IF ConveyorHasFault OR NOT SystemSafety.Safety_SystemEstopsOK THEN
	// Red light SOLID ON
	GVL_IO.LT_7221_Red := TRUE;
ELSE
	IF ConveyorHasWarn THEN
		// Orange Light SOLID ON
		GVL_IO.LT_7241_Yellow := TRUE;
	ELSE
		IF ConveyorInAuto THEN
			// Green Light SOLID ON
			GVL_IO.LT_7271_Green := TRUE;
		ELSE
			GVL_IO.LT_7271_Green := SysShrtPulseTmr.Output;
		END_IF
	END_IF
	IF GVL_IO.HornMainPanel THEN
		// Orange Light FLASHING ON
		GVL_IO.LT_7241_Yellow := SysShrtPulseTmr.Output;
	END_IF;
END_IF

// Initialise the Stack Light, only changing values as required
GVL_IO.LT_12161_Green := FALSE;
GVL_IO.LT_12131_Yellow := FALSE;
GVL_IO.LT_12121_Red := FALSE;
	
IF ConveyorHasFault OR NOT SystemSafety.Safety_SystemEstopsOK THEN
	// Red light SOLID ON
	GVL_IO.LT_12121_Red := TRUE;
ELSE
	IF ConveyorHasWarn THEN
		// Orange Light SOLID ON
		GVL_IO.LT_12131_Yellow := TRUE;
	ELSE
		IF ConveyorInAuto THEN
			// Green Light SOLID ON
			GVL_IO.LT_12161_Green := TRUE;
		ELSE
			GVL_IO.LT_12161_Green := SysShrtPulseTmr.Output;
		END_IF
	END_IF
	IF GVL_IO.HornMainPanel THEN
		// Orange Light FLASHING ON
		GVL_IO.LT_12131_Yellow := SysShrtPulseTmr.Output;
	END_IF;
END_IF

END_PROGRAM

// ---- POUs/FunctionBlocks/Utils/FB_SystemCntrl.TcPOU
FUNCTION_BLOCK FB_SystemCntrl

(* System Interlock and Event Set up,
	Uses Interlocks.
	Doesn't use Start Conditions or the horn delay  
	Uses Events
	
	This exists to allow the Interlock/Event descriptions and setup to be managed through the HMI
	and be easily setup as system faults.
*)
VAR_IN_OUT
	Sts_EquipState				: ST_EquipmentStatus;		// State Status
END_VAR
VAR_INPUT
	{attribute 'OPC.UA.DA' := '1'}
	In_o_EquipStatePB			: ST_StateCntrlPB;		// Hmi push buttons to change states
	In_p_EquipStatePB			: ST_StateCntrlPB;		// Other push buttons to change states
	{attribute 'OPC.UA.DA' := '1'}
	Cfg_EquipLabel				: STRING(20);		// Label of the equipment
	// Events
	In_SystemEvents				: UINT;		// Event that is specific to the instance of the solenoid/actuator
	Cfg_EquipEvntsArry			: ARRAY [0..15] OF ST_CfgEvents;
	
	// Interlocks that can be Instance Specific
	In_SystemIntlks				: UINT;		// Interlock that is specific to the instance of the solenoid/actuator
	Cfg_EquipIntlksArry		: ARRAY [0..15] OF ST_CfgEvents;		// Descriptions of the Interlock 
	
END_VAR
VAR_OUTPUT
	{attribute 'OPC.UA.DA' := '1'}
	Out_Auto					:	BOOL;	// Combine HMI and Other Start/Auto signals to issue a single START/AUTO command
	{attribute 'OPC.UA.DA' := '1'}
	Out_Stop					:	BOOL;	// Combine HMI and Other Stop signals to issue a single STOP command
	{attribute 'OPC.UA.DA' := '1'}
	Out_Reset					:	BOOL;	// Combine HMI and Other Reset signals to issue a single RESET command
	{attribute 'OPC.UA.DA' := '1'}
	Sts_All_Intlks_OK			: BOOL;		// Status bit to show that all interloks are good to Run 
	{attribute 'OPC.UA.DA' := '1'}
	Sts_FaultActive				: BOOL;	// Status Bit Showing that a fault is present (0= No Active Faults, 1= Fault Active)
	{attribute 'OPC.UA.DA' := '1'}
	Sts_WarnActive				: BOOL;	// Status Bit Showing that a warning is present (0= No Active Warnings, 1= Warning Active)
	{attribute 'OPC.UA.DA' := '1'}
	Sts_All_Evnts_OK			: BOOL;		// Status Bit Showing that ALL Events are OK to RUN (0= Event Present, 1= OK to Run)
	{attribute 'OPC.UA.DA' := '1'}
	Sts_IntlksArry				: ARRAY[0..15] OF ST_EventSts;		// Interlock status 0 to 15 Input
	{attribute 'OPC.UA.DA' := '1'}
	Sts_FaultsArry				: ARRAY[0..15] OF ST_EventSts;	// Status of each Fault Event State (0= OFF, 1=ON)
	{attribute 'OPC.UA.DA' := '1'}
	Sts_WarnsArry				: ARRAY[0..15] OF ST_EventSts;		// Status of each Warning Event State (0= OFF, 1=ON)
	{attribute 'OPC.UA.DA' := '1'}
	Sts_EvntsArry				: ARRAY[0..15] OF ST_EventSts; 	// Status of each Event State (0= OFF, 1=ON)
END_VAR
VAR
	System_fbIntrlks				: FB_Intlks_Latch;
	System_IntlksArry				: ARRAY[0..15] OF BOOL;
	System_EventManager				: FB_EventMngr;
	System_EventArry				: ARRAY[0..15] OF BOOL;
	System_LatchIgnore				: BOOL := FALSE;		// Put as a place holder for ease of future use
	System_LatchReset				: BOOL := FALSE;		//Put as a place holder for ease of future use
	System_IntlkBypassed			: ARRAY [0..15] OF BOOL;		//Put as a place holder for ease of future use
END_VAR

// Set Up inputs for interlocks that are specific for the configuration instance
System_IntlksArry[0] := In_SystemIntlks.0;
System_IntlksArry[1] := In_SystemIntlks.1; 
System_IntlksArry[2] := In_SystemIntlks.2;
System_IntlksArry[3] := In_SystemIntlks.3;
System_IntlksArry[4] := In_SystemIntlks.4;
System_IntlksArry[5] := In_SystemIntlks.5;
System_IntlksArry[6] := In_SystemIntlks.6;
System_IntlksArry[7] := In_SystemIntlks.7;
System_IntlksArry[8] := In_SystemIntlks.8;
System_IntlksArry[9] := In_SystemIntlks.9; 
System_IntlksArry[10] := In_SystemIntlks.10;
System_IntlksArry[11] := In_SystemIntlks.11;
System_IntlksArry[12] := In_SystemIntlks.12;
System_IntlksArry[13] := In_SystemIntlks.13;
System_IntlksArry[14] := In_SystemIntlks.14;
System_IntlksArry[15] := In_SystemIntlks.15;
	
// Call Interlock block
System_fbIntrlks(
	In_Intlks:= System_IntlksArry,
	CFG_IntlksArry:= Cfg_EquipIntlksArry, 
	HMI_LatchIgnore:= System_LatchIgnore, 
	HMI_LatchReset:= System_LatchReset, 
	All_Intlk_OK=> Sts_All_Intlks_OK, 
	STS_Intlks=> Sts_IntlksArry);
	
System_EventArry[0]:= In_SystemEvents.0;
System_EventArry[1]:= In_SystemEvents.1;
System_EventArry[2]:= In_SystemEvents.2;
System_EventArry[3]:= In_SystemEvents.3;
System_EventArry[4]:= In_SystemEvents.4;
System_EventArry[5]:= In_SystemEvents.5;
System_EventArry[6]:= In_SystemEvents.6;
System_EventArry[7]:= In_SystemEvents.7;
System_EventArry[8]:= In_SystemEvents.8;
System_EventArry[9]:= In_SystemEvents.9;
System_EventArry[10]:= In_SystemEvents.10;
System_EventArry[11]:= In_SystemEvents.11;
System_EventArry[12]:= In_SystemEvents.12;
System_EventArry[13]:= In_SystemEvents.13;
System_EventArry[14]:= In_SystemEvents.14;
System_EventArry[15]:= In_SystemEvents.15;

// Event Manager
System_EventManager(
	sEquipStateCntrlSts := Sts_EquipState.Sts_EquipmentState,
	In_EventsArry := System_EventArry ,  
	CFG_EvntsArry:= Cfg_EquipEvntsArry, 
	HMI_LatchReset:= In_o_EquipStatePB.ResetPB OR In_p_EquipStatePB.ResetPB,
	Out_FaultActive=> Sts_FaultActive, 
	Out_WarnActive=> Sts_WarnActive, 
	Sts_All_Evnts_OK=> Sts_All_Evnts_OK, 
	Sts_FaultsArry=> Sts_FaultsArry, 
	Sts_WarnsArry=> Sts_WarnsArry, 
	Sts_EvntsArry=> Sts_EvntsArry);

// Activate the Out_ variables
Out_Auto := In_o_EquipStatePB.AutoPB OR In_p_EquipStatePB.AutoPB;
Out_Stop := In_o_EquipStatePB.StopPB OR In_p_EquipStatePB.StopPB;
Out_Reset := In_o_EquipStatePB.ResetPB OR In_p_EquipStatePB.ResetPB;

// Populate the Sts Output Variables
Sts_EquipState.Sts_EquipmentState.CrntState := 1;
Sts_EquipState.Sts_All_Intlks_OK  := Sts_All_Intlks_OK;
Sts_EquipState.Sts_All_Evnts_OK  := Sts_All_Evnts_OK;
Sts_EquipState.Sts_FaultActive := Sts_FaultActive;
Sts_EquipState.Sts_WarnActive := Sts_WarnActive;

END_FUNCTION_BLOCK

// ---- POUs/SystemSafety.TcPOU
PROGRAM SystemSafety
VAR
	{attribute 'OPC.UA.DA' := '1'}
	System_SafetyState : ST_SafetyState;
	{attribute 'OPC.UA.DA' := '1'}

	{attribute 'OPC.UA.DA' := '1'}
	Safety_SystemEstopsOK AT %I* : BOOL;
	{attribute 'OPC.UA.DA' := '1'}
	Safety_PanelEstop AT %I* : BOOL;
	{attribute 'OPC.UA.DA' := '1'}
	ZoneSafe_EDM AT %I*: BOOL; 
	{attribute 'OPC.UA.DA' := '1'}
	SecondFloorShaft_Estop_OK AT %I* : BOOL;
	{attribute 'OPC.UA.DA' := '1'}
	ThirdFloorShaft_Estop_OK AT %I* : BOOL;
END_VAR

// Set System Safety Variables 
System_SafetyState.ErrAck := System.Safety_Reset;
System_SafetyState.CommErrAck := System.Safety_Reset;
System_SafetyState.Reset := System.Safety_Reset;
System_SafetyState.Run := TRUE;

END_PROGRAM

// ---- POUs/FunctionBlocks/VFD/Functions/VFD.TcPOU
FUNCTION_BLOCK VFD
FUNCTION_BLOCK VFD
VAR_INPUT
	RunVelocity				: INT;
	RunRequest				: BOOL;
	PLCFault				: BOOL;
	Reset					: BOOL;
	VelocityThreshold		: INT;
END_VAR
VAR_OUTPUT
	ActualVelocity 	AT %I* 	: INT;
	StatusWord		AT %I* 	: UINT;
	Run_OK					: BOOL;
	STO_Active				: BOOL;
	IsRunning				: BOOL;
	IsFaulted 				: BOOL;
END_VAR
VAR
	VFD_State				: DriveState;
	ControlWord 	AT %Q* 	: UINT;
	TargetVelocity 	AT %Q*	: INT;
	StatusWordFiltered		: UINT;
END_VAR
VAR CONSTANT
	SAFETY_TORQUE_OFF_ACTIVE : INT := 15;
END_VAR

StatusWordFiltered := StatusWord AND 16#006F;

VFD_State(StatusWord := StatusWordFiltered, Run_Drive := RunRequest, ControlWord => ControlWord, PLCFault := PLCFault, ResetFault := Reset);

IF Reset THEN
	Reset := FALSE;
END_IF

Run_OK := (StatusWordFiltered = Drive_State.READY_TO_SWITCH_ON) OR (StatusWordFiltered = Drive_State.SWITCHED_ON) OR (StatusWordFiltered = Drive_State.OPERATION_ENABLED);

IF StatusWordFiltered = Drive_State.OPERATION_ENABLED THEN
	TargetVelocity := RunVelocity;
ELSE
	TargetVelocity := 0;	
END_IF

STO_Active := StatusWord.SAFETY_TORQUE_OFF_ACTIVE;
 
IsRunning := ActualVelocity >= VelocityThreshold;
IsFaulted := VFD_State.Fault;

END_FUNCTION_BLOCK

// ---- POUs/CommStatus.TcPOU
PROGRAM CommStatus
VAR
	In_Dummy		:	BOOL;	// Replace per function call with IO point

	DebounceOnTime:	TIME := T#500MS;     // Default Value	
	DebounceOffTime:	TIME := T#1S;     // Default Value
		
	RIO1181_CommFault: FB_DigDebnce;	// Remote IO Block 1181 Communication Fault
	RIO4172_CommFault: FB_DigDebnce;	// Remote IO Block 4172 Communication Fault
	RIO5151_CommFault: FB_DigDebnce;	// Remote IO Block 5151 Communication Fault
	RIO6171_CommFault: FB_DigDebnce;	// Remote IO Block 6171 Communication Fault
	RIO7161_CommFault: FB_DigDebnce;	// Remote IO Block 7161 Communication Fault
	RIO8181_CommFault: FB_DigDebnce;	// Remote IO Block 8181 Communication Fault
	RIO11141_CommFault: FB_DigDebnce;	// Remote IO Block 11141 Communication Fault	
	RIO12171_CommFault: FB_DigDebnce;	// Remote IO Block 12171 Communication Fault
	RIO15181_CommFault: FB_DigDebnce;	// Remote IO Block 15181 Communication Fault
	RIO16171_CommFault: FB_DigDebnce;	// Remote IO Block 16171 Communication Fault
	
	BCR_S6040_01_CommFault: FB_DigDebnce;;		// Bar Code Reader 6040_01 Communication Fault
	BCR_S7004_01_CommFault: FB_DigDebnce;;		// Bar Code Reader 7004_01 Communication Fault
	
	Ethernet_CommFault: FB_DigDebnce;;		// Ethernet Adapter Status Communication Fault
	
END_VAR

// Remote IO Blocks --------------------
RIO1181_CommFault(
	In:= GVL_IO.RIO1181_WcState, 
	CFG_OKState:= 0, 
	CFG_OnDlyTime:= DebounceOnTime, 
	CFG_OffDlyTime:= DebounceOffTime, 
	In_Sim:= , 
	);
	
RIO4172_CommFault(
	In:= GVL_IO.RIO4172_WcState, 
	CFG_OKState:= 0, 
	CFG_OnDlyTime:= DebounceOnTime, 
	CFG_OffDlyTime:= DebounceOffTime, 
	In_Sim:= , 
	);

RIO5151_CommFault(
	In:= GVL_IO.RIO5151_WcState, 
	CFG_OKState:= 0, 
	CFG_OnDlyTime:= DebounceOnTime, 
	CFG_OffDlyTime:= DebounceOffTime, 
	In_Sim:= , 
	);

RIO6171_CommFault(
	In:= GVL_IO.RIO6171_WcState, 
	CFG_OKState:= 0, 
	CFG_OnDlyTime:= DebounceOnTime, 
	CFG_OffDlyTime:= DebounceOffTime, 
	In_Sim:= , 
	);
	
RIO7161_CommFault(
	In:= GVL_IO.RIO7161_WcState, 
	CFG_OKState:= 0, 
	CFG_OnDlyTime:= DebounceOnTime, 
	CFG_OffDlyTime:= DebounceOffTime, 
	In_Sim:= , 
	);
	
RIO8181_CommFault(
	In:= GVL_IO.RIO8181_WcState, 
	CFG_OKState:= 0, 
	CFG_OnDlyTime:= DebounceOnTime, 
	CFG_OffDlyTime:= DebounceOffTime, 
	In_Sim:= , 
	);
	
RIO11141_CommFault(
	In:= GVL_IO.RIO11141_WcState, 
	CFG_OKState:= 0, 
	CFG_OnDlyTime:= DebounceOnTime, 
	CFG_OffDlyTime:= DebounceOffTime, 
	In_Sim:= , 
	);
	
RIO11141_CommFault(
	In:= GVL_IO.RIO11141_WcState, 
	CFG_OKState:= 0, 
	CFG_OnDlyTime:= DebounceOnTime, 
	CFG_OffDlyTime:= DebounceOffTime, 
	In_Sim:= , 
	);
	
RIO12171_CommFault(
	In:= GVL_IO.RIO12171_WcState, 
	CFG_OKState:= 0, 
	CFG_OnDlyTime:= DebounceOnTime, 
	CFG_OffDlyTime:= DebounceOffTime, 
	In_Sim:= , 
	);
	
RIO15181_CommFault(
	In:= GVL_IO.RIO15181_WcState, 
	CFG_OKState:= 0, 
	CFG_OnDlyTime:= DebounceOnTime, 
	CFG_OffDlyTime:= DebounceOffTime, 
	In_Sim:= , 
	);
	
RIO16171_CommFault(
	In:= GVL_IO.RIO16171_WcState, 
	CFG_OKState:= 0, 
	CFG_OnDlyTime:= DebounceOnTime, 
	CFG_OffDlyTime:= DebounceOffTime, 
	In_Sim:= , 
	);

// Bar Code Readers --------------------	
BCR_S6040_01_CommFault(
	In:= BarCodeReaders.BCR_S6040_01.Out_DeviceState = 0, 
	CFG_OKState:= 1, 
	CFG_OnDlyTime:= DebounceOnTime, 
	CFG_OffDlyTime:= DebounceOffTime, 
	In_Sim:= , 
	);
BCR_S7004_01_CommFault(
	In:= BarCodeReaders.BCR_S7004_01.Out_DeviceState = 0, 
	CFG_OKState:= 1, 
	CFG_OnDlyTime:= DebounceOnTime, 
	CFG_OffDlyTime:= DebounceOffTime, 
	In_Sim:= , 
	);
	
// Ethernet Controller	
Ethernet_CommFault(
	In:= GVL_IO.EthernetAdapter_State = 0, 
	CFG_OKState:= 1, 
	CFG_OnDlyTime:= DebounceOnTime, 
	CFG_OffDlyTime:= DebounceOffTime, 
	In_Sim:= , 
	);

END_PROGRAM

// ---- POUs/FunctionBlocks/Utils/Filters/FB_DigDebnce.TcPOU
(*
Function Block to filter the ON and OFF of a digital input In
The normal OK state can be configured with CFG_OKState
The Times for the On and Off delays are configured by CFG_OnDlyTime and CFG_OffDlyTime
and can be simulated using the In_Sim input
If the input In goes true the output OutOnFltrd is set to true after the on delay time has elapsed
If the input In goes false the output CFG_OffDlyTime will be held on until the off delay time has elapsed
The output OutOnOffFltrd is delayed for both on and off as described above
The status outputs Sts_OnDlyActive and Sts_OffDlyActive show that the delays are active
*)
FUNCTION_BLOCK FB_DigDebnce
VAR_INPUT
	In:	BOOL;	// Digital Input
	CFG_OKState:	BOOL;		// The OK or ON State of the Input (0 or 1)
	CFG_OnDlyTime:	TIME;		// Time to delay Output turning On after Input is On
	CFG_OffDlyTime:	TIME;		// Time to delay Output turning Off after Input is Off
	In_Sim:	BOOL;		// Simulation Input Bit acts just like the input but can be forced from the program for testing
END_VAR
VAR_OUTPUT
	{attribute 'OPC.UA.DA' := '1'}
	Out:	BOOL;		// Output Based on ON or OK state
	OutOnFltrd:	BOOL;		// ON filtered Only Output
	OutOffFltrd:	BOOL;		// Off filtered Only OutPut
	OutOnOffFltrd:	BOOL;		// Both On and Off Filtered Output 
	Sts_OnDlyActive: BOOL;
	Sts_OffDlyActive: BOOL;
	Sts_OnOffDlyActive: BOOL;
END_VAR
VAR
	OnDly_Ton: TON;
	OffDlyTof: TOF;
	OnOffDlyTof: TOF;
	OnOffDly_SR: SR;
	
END_VAR

// Compare to normal ON state
Out := (In OR In_Sim) XOR CFG_OKState;

// Setup On Delay
OnDly_Ton(IN:= Out, PT:= CFG_OnDlyTime , Q=> OutOnFltrd , ET=> );
Sts_OnDlyActive := Out <> OutOnFltrd;

//Setup Off Delay
OffDlyTof(IN:= Out , PT:= CFG_OffDlyTime , Q=> OutOffFltrd , ET=> );
Sts_OffDlyActive := Out <> OutOffFltrd;

//Setup Both On and Off Delayed
//OnOffDlyTof(IN:= OutOnFltrd , PT:= CFG_OffDlyTime , Q=> OutOnOffFltrd , ET=> );
OnOffDly_SR(SET1 := OutOnFltrd, RESET := (NOT OffDlyTof.Q), Q1 => OutOnOffFltrd);
Sts_OnOffDlyActive := Out <> OutOnOffFltrd;

END_FUNCTION_BLOCK

// ---- POUs/ProxSensors.TcPOU
PROGRAM ProxSensors
VAR
	DebounceOnTime:	TIME := T#5MS;     // Default Value
	DebounceOffTime:	TIME := T#500MS;     // Default Value
	JamDetectTime:	TIME := T#5S;     // Default Value

	
	In_PX_1281_Extended AT %I* : BOOL;      // Mapped IO input for PX
	PX_1281_Extended:  FB_DigDebnce;		// P6020 POWER TRANSFER EXTENDED PROX
//----------------------------------------GR6040_01--------------------------------------------------------------
	In_PX_6241_Retracted AT %I* : BOOL;      // Mapped IO input for PX
	PX_6241_Retracted:  FB_DigDebnce;		// GR6040-01 "D" GRIPPER RETRACTED PROX

	In_PX_6261_Extended AT %I* : BOOL;      // Mapped IO input for PX
	PX_6261_Extended:  FB_DigDebnce;		// GR6040-01 "D" GRIPPER EXTENDED PROX
//----------------------------------------GR6040_02--------------------------------------------------------------
	In_PX_6121_Retracted AT %I* : BOOL;      // Mapped IO input for PX
	PX_6121_Retracted:  FB_DigDebnce;		// GR6040-02 "D" GRIPPER RETRACTED PROX

	In_PX_6151_Extended AT %I* : BOOL;      // Mapped IO input for PX
	PX_6151_Extended:  FB_DigDebnce;		// GR6040-02 "D" GRIPPER EXTENDED PROX
//----------------------------------------PI6040_01--------------------------------------------------------------
	In_PX_6122_Retracted AT %I* : BOOL;      // Mapped IO input for PX
	PX_6122_Retracted:  FB_DigDebnce;		// PI6040-01 "D" GRIPPER RETRACTED PROX

	In_PX_6152_Extended AT %I* : BOOL;      // Mapped IO input for PX
	PX_6152_Extended:  FB_DigDebnce;		// PI6040-01 "D" GRIPPER EXTENDED PROX
//----------------------------------------PU6040_01--------------------------------------------------------------
	In_PX_7271_Retracted AT %I* : BOOL;      // Mapped IO input for PX
	PX_7271_Retracted:  FB_DigDebnce;		// PU6040-01 PUSH DIVERT RETRACTED PROX

	In_PX_7301_Extended AT %I* : BOOL;      // Mapped IO input for PX
	PX_7301_Extended:  FB_DigDebnce;		// PU6040-01 PUSH DIVERT EXTENDED PROX
//----------------------------------------PU6040_02--------------------------------------------------------------
	In_PX_7122_Retracted AT %I* : BOOL;      // Mapped IO input for PX
	PX_7122_Retracted:  FB_DigDebnce;		// PU6040-02 PUSH DIVERT RETRACTED PROX

	In_PX_7151_Extended AT %I* : BOOL;      // Mapped IO input for PX
	PX_7151_Extended:  FB_DigDebnce;		// PU6040-02 PUSH DIVERT EXTENDED PROX
//----------------------------------------PU6040_03--------------------------------------------------------------
	In_PX_8321_Retracted AT %I* : BOOL;      // Mapped IO input for PX
	PX_8321_Retracted:  FB_DigDebnce;		// PU6040-03 PUSH DIVERT RETRACTED PROX

	In_PX_8291_Extended AT %I* : BOOL;      // Mapped IO input for PX
	PX_8291_Extended:  FB_DigDebnce;		// PU6040-03 PUSH DIVERT EXTENDED PROX
//----------------------------------------PU6040_04--------------------------------------------------------------	
	In_PX_8091_Retracted AT %I* : BOOL;      // Mapped IO input for PX
	PX_8091_Retracted:  FB_DigDebnce;		// PU6040-04 PUSH DIVERT RETRACTED PROX

	In_PX_8121_Extended AT %I* : BOOL;      // Mapped IO input for PX
	PX_8121_Extended:  FB_DigDebnce;		// PU6040-04 PUSH DIVERT EXTENDED PROX

//------------------------------------------------------------------------------------------------------
	In_PX_16231_Extended AT %I* : BOOL;      // Mapped IO input for PX
	PX_16231_Extended:  FB_DigDebnce;		// P7035 POWER TRANSFER EXTENDED PROX

END_VAR

//----------------------------------------P6020--------------------------------------------------------------
// P6020 POWER TRANSFER Extended
PX_1281_Extended(
	In:= In_PX_1281_Extended,
	CFG_OKState:= 0,
	CFG_OnDlyTime:= DebounceOnTime,
	CFG_OnDlyTime:= DebounceOffTime,
	In_Sim:= 
	);
//----------------------------------------GR6040_01--------------------------------------------------------------
// GR6040-01 "D" GRIPPER Retracted
PX_6241_Retracted(
	In:= In_PX_6241_Retracted,
	CFG_OKState:= 0,
	CFG_OnDlyTime:= DebounceOnTime,
	CFG_OnDlyTime:= DebounceOffTime,
	In_Sim:= 
	);

// GR6040-01 "D" GRIPPER Extended
PX_6261_Extended(
	In:= In_PX_6261_Extended,
	CFG_OKState:= 0,
	CFG_OnDlyTime:= DebounceOnTime,
	CFG_OnDlyTime:= DebounceOffTime,
	In_Sim:= 
	);
//----------------------------------------GR6040_02--------------------------------------------------------------
// GR6040-02 "D" GRIPPER Retracted
PX_6121_Retracted(
	In:= In_PX_6121_Retracted,
	CFG_OKState:= 0,
	CFG_OnDlyTime:= DebounceOnTime,
	CFG_OnDlyTime:= DebounceOffTime,
	In_Sim:= 
	);

// GR6040-02 "D" GRIPPER Extended
PX_6151_Extended(
	In:= In_PX_6151_Extended,
	CFG_OKState:= 0,
	CFG_OnDlyTime:= DebounceOnTime,
	CFG_OnDlyTime:= DebounceOffTime,
	In_Sim:= 
	);
//----------------------------------------PI6040_01--------------------------------------------------------------
// PI6040-01 "D" GRIPPER Retracted
PX_6122_Retracted(
	In:= In_PX_6122_Retracted,
	CFG_OKState:= 0,
	CFG_OnDlyTime:= DebounceOnTime,
	CFG_OnDlyTime:= DebounceOffTime,
	In_Sim:= 
	);

// PI6040-01 "D" GRIPPER Extended
PX_6152_Extended(
	In:= In_PX_6152_Extended,
	CFG_OKState:= 0,
	CFG_OnDlyTime:= DebounceOnTime,
	CFG_OnDlyTime:= DebounceOffTime,
	In_Sim:= 
	);
//----------------------------------------PU6040_01--------------------------------------------------------------
// PU6040-01 PUSH DIVERT Retracted
PX_7271_Retracted(
	In:= In_PX_7271_Retracted,
	CFG_OKState:= 0,
	CFG_OnDlyTime:= DebounceOnTime,
	CFG_OnDlyTime:= DebounceOffTime,
	In_Sim:= 
	);

// PU6040-01 PUSH DIVERT Extended
PX_7301_Extended(
	In:= In_PX_7301_Extended,
	CFG_OKState:= 0,
	CFG_OnDlyTime:= DebounceOnTime,
	CFG_OnDlyTime:= DebounceOffTime,
	In_Sim:= 
	);
//----------------------------------------PU6040_02--------------------------------------------------------------
// PU6040-02 PUSH DIVERT Retracted
PX_7122_Retracted(
	In:= In_PX_7122_Retracted,
	CFG_OKState:= 0,
	CFG_OnDlyTime:= DebounceOnTime,
	CFG_OnDlyTime:= DebounceOffTime,
	In_Sim:= 
	);

// PU6040-02 PUSH DIVERT Extended
PX_7151_Extended(
	In:= In_PX_7151_Extended,
	CFG_OKState:= 0,
	CFG_OnDlyTime:= DebounceOnTime,
	CFG_OnDlyTime:= DebounceOffTime,
	In_Sim:= 
	);
//----------------------------------------PU6040_03--------------------------------------------------------------	
	// PU6040-03 PUSH DIVERT Retracted
PX_8321_Retracted(
	In:= In_PX_8321_Retracted,
	CFG_OKState:= 0,
	CFG_OnDlyTime:= DebounceOnTime,
	CFG_OnDlyTime:= DebounceOffTime,
	In_Sim:= 
	);

// PU6040-03 PUSH DIVERT Extended
PX_8291_Extended(
	In:= In_PX_8291_Extended,
	CFG_OKState:= 0,
	CFG_OnDlyTime:= DebounceOnTime,
	CFG_OnDlyTime:= DebounceOffTime,
	In_Sim:= 
	);
//----------------------------------------PU6040_04--------------------------------------------------------------
// PU6040-04 PUSH DIVERT Retracted
PX_8091_Retracted(
	In:= In_PX_8091_Retracted,
	CFG_OKState:= 0,
	CFG_OnDlyTime:= DebounceOnTime,
	CFG_OnDlyTime:= DebounceOffTime,
	In_Sim:= 
	);
	
// PU6040-04 PUSH DIVERT Extended
PX_8121_Extended(
	In:= In_PX_8121_Extended,
	CFG_OKState:= 0,
	CFG_OnDlyTime:= DebounceOnTime,
	CFG_OnDlyTime:= DebounceOffTime,
	In_Sim:= 
	);
//----------------------------------------P7035--------------------------------------------------------------
// P7035 POWER TRANSFER Extended
PX_16231_Extended(
	In:= In_PX_16231_Extended,
	CFG_OKState:= 0,
	CFG_OnDlyTime:= DebounceOnTime,
	CFG_OnDlyTime:= DebounceOffTime,
	In_Sim:= 
	);

END_PROGRAM

// ---- POUs/Solenoids.TcPOU
PROGRAM Solenoids

VAR
	 nEquipIndex:	DINT := 0;	// Dummy Equipment Index for Non reporting equipment
//----------------------------------------GR6040_02--------------------------------------------------------------
   cfgGR6040_02Label:	STRING(20) :=  'GR6040_02';
   cfgGR6040_02ExtendTODetectTime:	TIME := T#5S;
   cfgGR6040_02RetractTODetectTime:	TIME := T#5S;
   GR6040_02			: FB_Solenoid_SA;
   GR6040_02_StatePB	: ST_StateCntrlPB;
   GR6040_02_Status	: ST_EquipmentStatus;		// Gripper State 

//----------------------------------------GR6040_01--------------------------------------------------------------
   cfgGR6040_01Label:	STRING(20) :=  'GR6040_01';
   cfgGR6040_01ExtendTODetectTime:	TIME := T#5S;
   cfgGR6040_01RetractTODetectTime:	TIME := T#5S;
   GR6040_01			: FB_Solenoid_SA;
   GR6040_01_StatePB	: ST_StateCntrlPB;
   GR6040_01_Status	: ST_EquipmentStatus;		// Gripper State 

//----------------------------------------PI6040_01--------------------------------------------------------------
   cfgPI6040_01Label:	STRING(20) :=  'PI6040_01';
   cfgPI6040_01ExtendTODetectTime:	TIME := T#5S;
   cfgPI6040_01RetractTODetectTime:	TIME := T#5S;
   PI6040_01			: FB_Solenoid_DA;
   PI6040_01_StatePB	: ST_StateCntrlPB;
   PI6040_01_Status	: ST_EquipmentStatus;		// Gripper State 

//----------------------------------------PU6040_01--------------------------------------------------------------
   cfgPU6040_01Label:	STRING(20) :=  'PU6040_01';
   cfgPU6040_01ExtendTODetectTime:	TIME := T#5S;
   cfgPU6040_01RetractTODetectTime:	TIME := T#5S;
   PU6040_01			: FB_Solenoid_SA;
   PU6040_01_StatePB	: ST_StateCntrlPB;
   PU6040_01_Status	: ST_EquipmentStatus;		// Gripper State 

//----------------------------------------PU6040_02--------------------------------------------------------------
   cfgPU6040_02Label:	STRING(20) :=  'PU6040_02';
   cfgPU6040_02ExtendTODetectTime:	TIME := T#5S;
   cfgPU6040_02RetractTODetectTime:	TIME := T#5S;
   PU6040_02			: FB_Solenoid_SA;
   PU6040_02_StatePB	: ST_StateCntrlPB;
   PU6040_02_Status	: ST_EquipmentStatus;		// Gripper State 

//----------------------------------------PU6040_03--------------------------------------------------------------
   cfgPU6040_03Label:	STRING(20) :=  'PU6040_03';
   cfgPU6040_03ExtendTODetectTime:	TIME := T#5S;
   cfgPU6040_03RetractTODetectTime:	TIME := T#5S;
   PU6040_03			: FB_Solenoid_SA;
   PU6040_03_StatePB	: ST_StateCntrlPB;
   PU6040_03_Status	: ST_EquipmentStatus;		// Gripper State 

//----------------------------------------PU6040_04--------------------------------------------------------------
   cfgPU6040_04Label:	STRING(20) :=  'PU6040_04';
   cfgPU6040_04ExtendTODetectTime:	TIME := T#5S;
   cfgPU6040_04RetractTODetectTime:	TIME := T#5S;
   PU6040_04			: FB_Solenoid_SA;
   PU6040_04_StatePB	: ST_StateCntrlPB;
   PU6040_04_Status	: ST_EquipmentStatus;		// Gripper State 
		
END_VAR

VAR PERSISTENT
//----------------------------------------GR6040_02--------------------------------------------------------------
{attribute 'OPC.UA.DA' := '1'}
cfgGR6040_02IntlksArry: ARRAY [0..15] OF ST_CfgEvents := [
   (Description := 'Low Air' , DeviceLabel := 'P6040' , OKState := TRUE, StopCode := E_StopCodes.LowAir),
   (Description := 'System Interlocks OK' , DeviceLabel := 'SYSTEM', OKState := TRUE, StopCode := E_StopCodes.SystemStop),
   14(())];
{attribute 'OPC.UA.DA' := '1'}
cfgGR6040_02EvntsArry: ARRAY [0..15] OF ST_CfgEvents := [
   (Description := 'Extend To', DeviceLabel := 'GR6040_02', LatchRequired := TRUE, OKState := FALSE, FaultWarn:= TRUE, StopCode := E_StopCodes.ActuatorTO),
   (Description := 'Retract TO', DeviceLabel := 'GR6040_02', LatchRequired := TRUE, FaultWarn:= TRUE, OKState := FALSE, StopCode := E_StopCodes.ActuatorTO),
   (Description := 'System Fault', DeviceLabel := '', OKState := TRUE, FaultWarn:= TRUE, StopCode := E_StopCodes.SystemStop),
   (Description := 'Low Air', DeviceLabel := 'P6040', OKState := TRUE, FaultWarn:= TRUE, StopCode := E_StopCodes.LowAir, EventDelay := T#100MS),
   (Description := 'System Estop', DeviceLabel := 'System', OKState := TRUE, FaultWarn:= TRUE, StopCode := E_StopCodes.SystemStop),
   (Description := 'RIO4172 Comm Fault', DeviceLabel := 'RIO4172', OKState := TRUE, FaultWarn:= TRUE, StopCode := E_StopCodes.FieldIOFLT),
   10(())];
//----------------------------------------GR6040_01--------------------------------------------------------------
{attribute 'OPC.UA.DA' := '1'}
cfgGR6040_01IntlksArry: ARRAY [0..15] OF ST_CfgEvents := [
   (Description := 'Low Air' , DeviceLabel := 'P6040' , OKState := TRUE, StopCode := E_StopCodes.LowAir),
   (Description := 'System Interlocks OK' , DeviceLabel := 'SYSTEM', OKState := TRUE, StopCode := E_StopCodes.SystemStop),
   14(())];
{attribute 'OPC.UA.DA' := '1'}
cfgGR6040_01EvntsArry: ARRAY [0..15] OF ST_CfgEvents := [
   (Description := 'Extend To', DeviceLabel := 'GR6040_01', LatchRequired := TRUE, OKState := FALSE, FaultWarn:= TRUE, StopCode := E_StopCodes.ActuatorTO),
   (Description := 'Retract TO', DeviceLabel := 'GR6040_01', LatchRequired := TRUE, FaultWarn:= TRUE, OKState := FALSE, StopCode := E_StopCodes.ActuatorTO),
   (Description := 'System Fault', DeviceLabel := '', OKState := TRUE, FaultWarn:= TRUE, StopCode := E_StopCodes.SystemStop),
   (Description := 'Low Air', DeviceLabel := 'P6040', OKState := TRUE, FaultWarn:= TRUE, StopCode := E_StopCodes.LowAir, EventDelay := T#100MS),
   (Description := 'System Estop', DeviceLabel := 'System', OKState := TRUE, FaultWarn:= TRUE, StopCode := E_StopCodes.SystemStop),
   (Description := 'RIO4172 Comm Fault', DeviceLabel := 'RIO4172', OKState := TRUE, FaultWarn:= TRUE, StopCode := E_StopCodes.FieldIOFLT),
   10(())];
//----------------------------------------PI6040_01--------------------------------------------------------------
{attribute 'OPC.UA.DA' := '1'}
cfgPI6040_01IntlksArry: ARRAY [0..15] OF ST_CfgEvents := [
   (Description := 'Low Air' , DeviceLabel := 'P6040' , OKState := TRUE, StopCode := E_StopCodes.LowAir),
   (Description := 'System Interlocks OK' , DeviceLabel := 'SYSTEM', OKState := TRUE, StopCode := E_StopCodes.SystemStop),
   14(())];
{attribute 'OPC.UA.DA' := '1'}
cfgPI6040_01EvntsArry: ARRAY [0..15] OF ST_CfgEvents := [
   (Description := 'Extend To', DeviceLabel := 'PI6040_01', LatchRequired := TRUE, OKState := FALSE, FaultWarn:= TRUE, StopCode := E_StopCodes.ActuatorTO),
   (Description := 'Retract TO', DeviceLabel := 'PI6040_01', LatchRequired := TRUE, FaultWarn:= TRUE, OKState := FALSE, StopCode := E_StopCodes.ActuatorTO),
   (Description := 'System Fault', DeviceLabel := '', OKState := TRUE, FaultWarn:= TRUE, StopCode := E_StopCodes.SystemStop),
   (Description := 'Low Air', DeviceLabel := 'P6040', OKState := TRUE, FaultWarn:= TRUE, StopCode := E_StopCodes.LowAir, EventDelay := T#100MS),
   (Description := 'System Estop', DeviceLabel := 'System', OKState := TRUE, FaultWarn:= TRUE, StopCode := E_StopCodes.SystemStop),
   (Description := 'RIO4172 Comm Fault', DeviceLabel := 'RIO4172', OKState := TRUE, FaultWarn:= TRUE, StopCode := E_StopCodes.FieldIOFLT),
   10(())];
//----------------------------------------PU6040_01--------------------------------------------------------------
{attribute 'OPC.UA.DA' := '1'}
cfgPU6040_01IntlksArry: ARRAY [0..15] OF ST_CfgEvents := [
   (Description := 'Low Air' , DeviceLabel := 'P6040' , OKState := TRUE, StopCode := E_StopCodes.LowAir),
   (Description := 'System Interlocks OK' , DeviceLabel := 'SYSTEM', OKState := TRUE, StopCode := E_StopCodes.SystemStop),
   (Description := 'Jam Detected' , DeviceLabel := 'PE_7151', OKState := TRUE, StopCode := E_StopCodes.ProductJam),
   13(())];
{attribute 'OPC.UA.DA' := '1'}
cfgPU6040_01EvntsArry: ARRAY [0..15] OF ST_CfgEvents := [
   (Description := 'Extend To', DeviceLabel := 'PU6040_01', LatchRequired := TRUE, OKState := FALSE, FaultWarn:= TRUE, StopCode := E_StopCodes.ActuatorTO),
   (Description := 'Retract TO', DeviceLabel := 'PU6040_01', LatchRequired := TRUE, FaultWarn:= TRUE, OKState := FALSE, StopCode := E_StopCodes.ActuatorTO),
   (Description := 'System Fault', DeviceLabel := '', OKState := TRUE, FaultWarn:= TRUE, StopCode := E_StopCodes.SystemStop),
   (Description := 'Low Air', DeviceLabel := 'P6040', OKState := TRUE, FaultWarn:= TRUE, StopCode := E_StopCodes.LowAir, EventDelay := T#100MS),
   (Description := 'System Estop', DeviceLabel := 'System', OKState := TRUE, FaultWarn:= TRUE, StopCode := E_StopCodes.SystemStop),
   (Description := 'RIO7161 Comm Fault', DeviceLabel := 'RIO7161', OKState := TRUE, FaultWarn:= TRUE, StopCode := E_StopCodes.FieldIOFLT),
   10(())];
//----------------------------------------PU6040_02--------------------------------------------------------------
{attribute 'OPC.UA.DA' := '1'}
cfgPU6040_02IntlksArry: ARRAY [0..15] OF ST_CfgEvents := [
   (Description := 'Low Air' , DeviceLabel := 'P6040' , OKState := TRUE, StopCode := E_StopCodes.LowAir),
   (Description := 'System Interlocks OK' , DeviceLabel := 'SYSTEM', OKState := TRUE, StopCode := E_StopCodes.SystemStop),
   (Description := 'Jam Detected' , DeviceLabel := 'PE_7211', OKState := TRUE, StopCode := E_StopCodes.ProductJam),
   12(())];
{attribute 'OPC.UA.DA' := '1'}
cfgPU6040_02EvntsArry: ARRAY [0..15] OF ST_CfgEvents := [
   (Description := 'Extend To', DeviceLabel := 'PU6040_02', LatchRequired := TRUE, OKState := FALSE, FaultWarn:= TRUE, StopCode := E_StopCodes.ActuatorTO),
   (Description := 'Retract TO', DeviceLabel := 'PU6040_02', LatchRequired := TRUE, FaultWarn:= TRUE, OKState := FALSE, StopCode := E_StopCodes.ActuatorTO),
   (Description := 'System Fault', DeviceLabel := '', OKState := TRUE, FaultWarn:= TRUE, StopCode := E_StopCodes.SystemStop),
   (Description := 'Low Air', DeviceLabel := 'P6040', OKState := TRUE, FaultWarn:= TRUE, StopCode := E_StopCodes.LowAir, EventDelay := T#100MS),
   (Description := 'System Estop', DeviceLabel := 'System', OKState := TRUE, FaultWarn:= TRUE, StopCode := E_StopCodes.SystemStop),
   (Description := 'RIO7161 Comm Fault', DeviceLabel := 'RIO7161', OKState := TRUE, FaultWarn:= TRUE, StopCode := E_StopCodes.FieldIOFLT),
   10(())];
//----------------------------------------PU6040_03--------------------------------------------------------------
{attribute 'OPC.UA.DA' := '1'}
cfgPU6040_03IntlksArry: ARRAY [0..15] OF ST_CfgEvents := [
   (Description := 'Low Air' , DeviceLabel := 'P6040' , OKState := TRUE, StopCode := E_StopCodes.LowAir),
   (Description := 'System Interlocks OK' , DeviceLabel := 'SYSTEM', OKState := TRUE, StopCode := E_StopCodes.SystemStop),
   (Description := 'Jam Detected' , DeviceLabel := 'PE_8141', OKState := TRUE, StopCode := E_StopCodes.ProductJam),
   13(())];
{attribute 'OPC.UA.DA' := '1'}
cfgPU6040_03EvntsArry: ARRAY [0..15] OF ST_CfgEvents := [
   (Description := 'Extend To', DeviceLabel := 'PU6040_03', LatchRequired := TRUE, OKState := FALSE, FaultWarn:= TRUE, StopCode := E_StopCodes.ActuatorTO),
   (Description := 'Retract TO', DeviceLabel := 'PU6040_03', LatchRequired := TRUE, FaultWarn:= TRUE, OKState := FALSE, StopCode := E_StopCodes.ActuatorTO),
   (Description := 'System Fault', DeviceLabel := '', OKState := TRUE, FaultWarn:= TRUE, StopCode := E_StopCodes.SystemStop),
   (Description := 'Low Air', DeviceLabel := 'P6040', OKState := TRUE, FaultWarn:= TRUE, StopCode := E_StopCodes.LowAir, EventDelay := T#100MS),
   (Description := 'System Estop', DeviceLabel := 'System', OKState := TRUE, FaultWarn:= TRUE, StopCode := E_StopCodes.SystemStop),
   (Description := 'RIO8181 Comm Fault', DeviceLabel := 'RIO8181', OKState := TRUE, FaultWarn:= TRUE, StopCode := E_StopCodes.FieldIOFLT),
   10(())];
//----------------------------------------PU6040_04--------------------------------------------------------------
{attribute 'OPC.UA.DA' := '1'}
cfgPU6040_04IntlksArry: ARRAY [0..15] OF ST_CfgEvents := [
   (Description := 'Low Air' , DeviceLabel := 'P6040' , OKState := TRUE, StopCode := E_StopCodes.LowAir),
   (Description := 'System Interlocks OK' , DeviceLabel := 'SYSTEM', OKState := TRUE, StopCode := E_StopCodes.SystemStop),
   (Description := 'Jam Detected' , DeviceLabel := 'PE_8181', OKState := TRUE, StopCode := E_StopCodes.ProductJam),
   13(())];
{attribute 'OPC.UA.DA' := '1'}
cfgPU6040_04EvntsArry: ARRAY [0..15] OF ST_CfgEvents := [
   (Description := 'Extend To', DeviceLabel := 'PU6040_04', LatchRequired := TRUE, OKState := FALSE, FaultWarn:= TRUE, StopCode := E_StopCodes.ActuatorTO),
   (Description := 'Retract TO', DeviceLabel := 'PU6040_04', LatchRequired := TRUE, FaultWarn:= TRUE, OKState := FALSE, StopCode := E_StopCodes.ActuatorTO),
   (Description := 'System Fault', DeviceLabel := '', OKState := TRUE, FaultWarn:= TRUE, StopCode := E_StopCodes.SystemStop),
   (Description := 'Low Air', DeviceLabel := 'P6040', OKState := TRUE, FaultWarn:= TRUE, StopCode := E_StopCodes.LowAir, EventDelay := T#100MS),
   (Description := 'System Estop', DeviceLabel := 'System', OKState := TRUE, FaultWarn:= TRUE, StopCode := E_StopCodes.SystemStop),
   (Description := 'RIO8181 Comm Fault', DeviceLabel := 'RIO8181', OKState := TRUE, FaultWarn:= TRUE, StopCode := E_StopCodes.FieldIOFLT),
   10(())];	
END_VAR

//!!!!!!!!!!!!!!!!!!!!CHange!!!!!!!!!!!!!!!!!!!!!!!!!!!!!!!!!!!!!
GVL_IO.SystemAirPressure := TRUE;



//----------------------------------------GR6040_01--------------------------------------------------------------
GR6040_01_StatePB.AutoPB := System.Cnvyr_Auto;
GR6040_01_StatePB.ManPB := System.Cnvyr_Manual;
GR6040_01_StatePB.ResetPB := System.Cnvyr_Reset;
GR6040_01_StatePB.OfflinePB := System.Cnvyr_Offline;
GR6040_01_StatePB.StopPB := System.Cnvyr_Manual;

// Initialize the Equipment Type
GR6040_01_Status.Sts_EquipmentState.EquipType := E_EquipType.Gripper_SA;

// Interlocks
GR6040_01.In_EquipIntlks.0:= GVL_IO.SystemAirPressure;

//Events
GR6040_01.In_EquipEvents.2:= System.SysEventsAllOk;
GR6040_01.In_EquipEvents.3:= GVL_IO.SystemAirPressure;
GR6040_01.In_EquipEvents.4:= SystemSafety.Safety_SystemEstopsOK;
GR6040_01.In_EquipEvents.5:= NOT CommStatus.RIO6171_CommFault.Out;

// Function Call
GR6040_01(
   In_p_EquipStatePB:= GR6040_01_StatePB,
   In_SimActive:= System.Sys_SimActive,
   Cfg_UseExtedFdbc:= FALSE,
   In_EquipInit:= GVL_IO.INIT,
   In_P_SVReqExtend:= Singulation_Control.SortSingulation.Out_Grabber_1_Ext,
   In_EquipRtrcdFdbck := ProxSensors.PX_6241_Retracted.OutOnFltrd,
   In_EquipExtdFdbck :=  ProxSensors.PX_6261_Extended.OutOnFltrd,
   Cfg_EquipIndex := nEquipIndex,
   Cfg_EquipLabel := cfgGR6040_01Label,
   Cfg_EquipDefState:= System.ConvDefaultState,
   Cfg_EquipIntlksArry:= cfgGR6040_01IntlksArry,
   Cfg_EquipEvntsArry:= cfgGR6040_01EvntsArry,
   Cfg_ExtendDetectTime:= cfgGR6040_01ExtendTODetectTime,
   Cfg_RetractDetectTime:= cfgGR6040_01RetractTODetectTime,
   Sts_EquipState := GR6040_01_Status,
   Out_ExtendCrntSV => GVL_IO.SV_6211_EXT ); 
//----------------------------------------GR6040_02--------------------------------------------------------------
GR6040_02_StatePB.AutoPB := System.Cnvyr_Auto;
GR6040_02_StatePB.ManPB := System.Cnvyr_Manual;
GR6040_02_StatePB.ResetPB := System.Cnvyr_Reset;
GR6040_02_StatePB.OfflinePB := System.Cnvyr_Offline;
GR6040_02_StatePB.StopPB := System.Cnvyr_Manual;

// Initialize the Equipment Type
GR6040_02_Status.Sts_EquipmentState.EquipType := E_EquipType.Gripper_SA;

// Interlocks
GR6040_02.In_EquipIntlks.0:= GVL_IO.SystemAirPressure;
//Events
GR6040_02.In_EquipEvents.2:= System.SysEventsAllOk;
GR6040_02.In_EquipEvents.3:= GVL_IO.SystemAirPressure;
GR6040_02.In_EquipEvents.4:= SystemSafety.Safety_SystemEstopsOK;
GR6040_02.In_EquipEvents.5:= NOT CommStatus.RIO6171_CommFault.Out;

// Function Call
GR6040_02(
   In_p_EquipStatePB:= GR6040_02_StatePB,
   In_SimActive:= System.Sys_SimActive,
   Cfg_UseExtedFdbc:= FALSE,
   In_EquipInit:= GVL_IO.INIT,
   In_P_SVReqExtend:= Singulation_Control.SortSingulation.Out_Grabber_2_Ext,
   In_EquipRtrcdFdbck := ProxSensors.PX_6121_Retracted.OutOnFltrd,
   In_EquipExtdFdbck := ProxSensors.PX_6151_Extended.OutOnFltrd,
   Cfg_EquipIndex := nEquipIndex,
   Cfg_EquipLabel := cfgGR6040_02Label,
   Cfg_EquipDefState:= System.ConvDefaultState,
   Cfg_EquipIntlksArry:= cfgGR6040_02IntlksArry,
   Cfg_EquipEvntsArry:= cfgGR6040_02EvntsArry,
   Cfg_ExtendDetectTime:= cfgGR6040_02ExtendTODetectTime,
   Cfg_RetractDetectTime:= cfgGR6040_02RetractTODetectTime,
   Sts_EquipState := GR6040_02_Status,
   Out_ExtendCrntSV => GVL_IO.SV_6181_EXT ); 

//----------------------------------------PI6040_01--------------------------------------------------------------
PI6040_01_StatePB.AutoPB := System.Cnvyr_Auto;
PI6040_01_StatePB.ManPB := System.Cnvyr_Manual;
PI6040_01_StatePB.ResetPB := System.Cnvyr_Reset;
PI6040_01_StatePB.OfflinePB := System.Cnvyr_Offline;
PI6040_01_StatePB.StopPB := System.Cnvyr_Manual;

// Initialize the Equipment Type
PI6040_01_Status.Sts_EquipmentState.EquipType := E_EquipType.Gripper_DA;

// Interlocks
PI6040_01.In_EquipIntlks.0:= GVL_IO.SystemAirPressure;
PI6040_01.In_EquipIntlks.2 :=(PI6040_01.In_P_SVReqExtend AND NOT PhotoEyes.PE_6241.Out) OR PI6040_01.In_P_SVReqRetract OR (NOT PhotoEyes.PE_6241.Out);
//Events
PI6040_01.In_EquipEvents.2:= System.SysEventsAllOk;
PI6040_01.In_EquipEvents.3:= GVL_IO.SystemAirPressure;
PI6040_01.In_EquipEvents.4:= SystemSafety.Safety_SystemEstopsOK;
PI6040_01.In_EquipEvents.5:= NOT CommStatus.RIO6171_CommFault.Out;

// Function Call
PI6040_01(
   In_p_EquipStatePB:= PI6040_01_StatePB,
   In_SimActive:= System.Sys_SimActive,
   In_EquipInit:= GVL_IO.INIT,
   In_P_SVReqExtend:= Singulation_Control.SortSingulation.Out_PinStop_Ext,
   In_P_SVReqRetract:= Singulation_Control.SortSingulation.Out_PinStop_Ret,
   In_EquipRtrcdFdbck := ProxSensors.PX_6122_Retracted.OutOnFltrd,
   In_EquipExtdFdbck :=  ProxSensors.PX_6152_Extended.OutOnFltrd,
   Cfg_EquipIndex := nEquipIndex,
   Cfg_EquipLabel := cfgPI6040_01Label,
   Cfg_EquipDefState:= System.ConvDefaultState,   Cfg_EquipIntlksArry:= cfgPI6040_01IntlksArry,
   Cfg_EquipEvntsArry:= cfgPI6040_01EvntsArry,
   Cfg_ExtendDetectTime:= cfgPI6040_01ExtendTODetectTime,
   Cfg_RetractDetectTime:= cfgPI6040_01RetractTODetectTime,
   Sts_EquipState := PI6040_01_Status,
   Out_ExtendCrntSV => GVL_IO.SV_6321_EXT,
   Out_RetractCrntSV => GVL_IO.SV_6301_RET);
//----------------------------------------PU6040_01--------------------------------------------------------------
PU6040_01_StatePB.AutoPB := System.Cnvyr_Auto;
PU6040_01_StatePB.ManPB := System.Cnvyr_Manual;
PU6040_01_StatePB.ResetPB := System.Cnvyr_Reset;
PU6040_01_StatePB.OfflinePB := System.Cnvyr_Offline;
PU6040_01_StatePB.StopPB := System.Cnvyr_Manual;

// Initialize the Equipment Type
PU6040_01_Status.Sts_EquipmentState.EquipType := E_EquipType.Gripper_SA;

// Interlocks
PU6040_01.In_EquipIntlks.0:= GVL_IO.SystemAirPressure;
PU6040_01.In_EquipIntlks.2:= Photoeyes.PE_7151.JamDetected;
//Events
PU6040_01.In_EquipEvents.2:= System.SysEventsAllOk;
PU6040_01.In_EquipEvents.3:= GVL_IO.SystemAirPressure;
PU6040_01.In_EquipEvents.4:= SystemSafety.Safety_SystemEstopsOK;
PU6040_01.In_EquipEvents.5:= NOT CommStatus.RIO7161_CommFault.Out;

// Function Call
PU6040_01(
   In_p_EquipStatePB:= PU6040_01_StatePB,
   In_SimActive:= System.Sys_SimActive,
   In_EquipInit:= GVL_IO.INIT,
   In_P_SVReqExtend:= Sorter.aSorterDiverts[1].Output1,
   In_EquipRtrcdFdbck := ProxSensors.PX_7271_Retracted.OutOnFltrd,
   In_EquipExtdFdbck :=  ProxSensors.PX_7301_Extended.OutOnFltrd,
   Cfg_EquipIndex := nEquipIndex,
   Cfg_EquipLabel := cfgPU6040_01Label,
   Cfg_EquipDefState:= System.ConvDefaultState,
   Cfg_EquipIntlksArry:= cfgPU6040_01IntlksArry,
   Cfg_EquipEvntsArry:= cfgPU6040_01EvntsArry,
   Cfg_ExtendDetectTime:= cfgPU6040_01ExtendTODetectTime,
   Cfg_RetractDetectTime:= cfgPU6040_01RetractTODetectTime,
   Sts_EquipState := PU6040_01_Status,
   Out_ExtendCrntSV => GVL_IO.SV_7121_EXT); 
//----------------------------------------PU6040_02--------------------------------------------------------------
PU6040_02_StatePB.AutoPB := System.Cnvyr_Auto;
PU6040_02_StatePB.ManPB := System.Cnvyr_Manual;
PU6040_02_StatePB.ResetPB := System.Cnvyr_Reset;
PU6040_02_StatePB.OfflinePB := System.Cnvyr_Offline;
PU6040_02_StatePB.StopPB := System.Cnvyr_Manual;

// Initialize the Equipment Type
PU6040_02_Status.Sts_EquipmentState.EquipType := E_EquipType.Gripper_SA;

// Interlocks
PU6040_02.In_EquipIntlks.0:= GVL_IO.SystemAirPressure;
PU6040_02.In_EquipIntlks.2:= Photoeyes.PE_7211.JamDetected;
//Events
PU6040_02.In_EquipEvents.2:= System.SysEventsAllOk;
PU6040_02.In_EquipEvents.3:= GVL_IO.SystemAirPressure;
PU6040_02.In_EquipEvents.4:= SystemSafety.Safety_SystemEstopsOK;
PU6040_02.In_EquipEvents.5:= NOT CommStatus.RIO7161_CommFault.Out;

// Function Call
PU6040_02(
   In_p_EquipStatePB:= PU6040_02_StatePB,
   In_SimActive:= System.Sys_SimActive,
   In_EquipInit:= GVL_IO.INIT,
   In_P_SVReqExtend:= Sorter.aSorterDiverts[2].Output1,
   In_EquipRtrcdFdbck := ProxSensors.PX_7122_Retracted.OutOnFltrd,
   In_EquipExtdFdbck :=  ProxSensors.PX_7151_Extended.OutOnFltrd,
   Cfg_EquipIndex := nEquipIndex,
   Cfg_EquipLabel := cfgPU6040_02Label,
   Cfg_EquipDefState:= System.ConvDefaultState,
   Cfg_EquipIntlksArry:= cfgPU6040_02IntlksArry,
   Cfg_EquipEvntsArry:= cfgPU6040_02EvntsArry,
   Cfg_ExtendDetectTime:= cfgPU6040_02ExtendTODetectTime,
   Cfg_RetractDetectTime:= cfgPU6040_02RetractTODetectTime,
   Sts_EquipState := PU6040_02_Status,
   Out_ExtendCrntSV => GVL_IO.SV_7181_EXT); 
//----------------------------------------PU6040_03--------------------------------------------------------------
PU6040_03_StatePB.AutoPB := System.Cnvyr_Auto;
PU6040_03_StatePB.ManPB := System.Cnvyr_Manual;
PU6040_03_StatePB.ResetPB := System.Cnvyr_Reset;
PU6040_03_StatePB.OfflinePB := System.Cnvyr_Offline;
PU6040_03_StatePB.StopPB := System.Cnvyr_Manual;

// Initialize the Equipment Type
PU6040_03_Status.Sts_EquipmentState.EquipType := E_EquipType.Gripper_SA;

// Interlocks
PU6040_03.In_EquipIntlks.0:= GVL_IO.SystemAirPressure;
PU6040_03.In_EquipIntlks.2:= Photoeyes.PE_8141.JamDetected;
//Events
PU6040_03.In_EquipEvents.2:= System.SysEventsAllOk;
PU6040_03.In_EquipEvents.3:= GVL_IO.SystemAirPressure;
PU6040_03.In_EquipEvents.4:= SystemSafety.Safety_SystemEstopsOK;
PU6040_03.In_EquipEvents.5:= NOT CommStatus.RIO8181_CommFault.Out;

// Function Call
PU6040_03(
   In_p_EquipStatePB:= PU6040_03_StatePB,
   In_SimActive:= System.Sys_SimActive,
   In_EquipInit:= GVL_IO.INIT,
   In_P_SVReqExtend:= Sorter.aSorterDiverts[3].Output1,
   In_EquipRtrcdFdbck := ProxSensors.PX_8321_Retracted.OutOnFltrd,
   In_EquipExtdFdbck :=  ProxSensors.PX_8291_Extended.OutOnFltrd,
   Cfg_EquipIndex := nEquipIndex,
   Cfg_EquipLabel := cfgPU6040_03Label,
   Cfg_EquipDefState:= System.ConvDefaultState,
   Cfg_EquipIntlksArry:= cfgPU6040_03IntlksArry,
   Cfg_EquipEvntsArry:= cfgPU6040_03EvntsArry,
   Cfg_ExtendDetectTime:= cfgPU6040_03ExtendTODetectTime,
   Cfg_RetractDetectTime:= cfgPU6040_03RetractTODetectTime,
   Sts_EquipState := PU6040_03_Status,
   Out_ExtendCrntSV => GVL_IO.SV_8111_EXT); 
//----------------------------------------PU6040_04--------------------------------------------------------------
PU6040_04_StatePB.AutoPB := System.Cnvyr_Auto;
PU6040_04_StatePB.ManPB := System.Cnvyr_Manual;
PU6040_04_StatePB.ResetPB := System.Cnvyr_Reset;
PU6040_04_StatePB.OfflinePB := System.Cnvyr_Offline;
PU6040_04_StatePB.StopPB := System.Cnvyr_Manual;

// Initialize the Equipment Type
PU6040_04_Status.Sts_EquipmentState.EquipType := E_EquipType.Gripper_SA;

// Interlocks
PU6040_04.In_EquipIntlks.0:= GVL_IO.SystemAirPressure;
PU6040_04.In_EquipIntlks.2:= Photoeyes.PE_8181.JamDetected;
//Events
PU6040_04.In_EquipEvents.2:= System.SysEventsAllOk;
PU6040_04.In_EquipEvents.3:= GVL_IO.SystemAirPressure;
PU6040_04.In_EquipEvents.4:= SystemSafety.Safety_SystemEstopsOK;
PU6040_04.In_EquipEvents.5:= NOT CommStatus.RIO8181_CommFault.Out;

// Function Call
PU6040_04(
   In_p_EquipStatePB:= PU6040_04_StatePB,
   In_SimActive:= System.Sys_SimActive,
   In_EquipInit:= GVL_IO.INIT,
   In_P_SVReqExtend:= Sorter.aSorterDiverts[4].Output1,
   In_EquipRtrcdFdbck := ProxSensors.PX_8091_Retracted.OutOnFltrd,
   In_EquipExtdFdbck :=  ProxSensors.PX_8121_Extended.OutOnFltrd,
   Cfg_EquipIndex := nEquipIndex,
   Cfg_EquipLabel := cfgPU6040_04Label,
   Cfg_EquipDefState:= System.ConvDefaultState,
   Cfg_EquipIntlksArry:= cfgPU6040_04IntlksArry,
   Cfg_EquipEvntsArry:= cfgPU6040_04EvntsArry,
   Cfg_ExtendDetectTime:= cfgPU6040_04ExtendTODetectTime,
   Cfg_RetractDetectTime:= cfgPU6040_04RetractTODetectTime,
   Sts_EquipState := PU6040_04_Status,
   Out_ExtendCrntSV => GVL_IO.SV_8161_EXT );

END_PROGRAM

// ---- POUs/FunctionBlocks/Solenoids/Functions/FB_Solenoid_SA.TcPOU
FUNCTION_BLOCK FB_Solenoid_SA

(* Single-Acting solenoid Set up,
	Uses Interlocks. No common interlocks
	Doesn't use Start Conditions or the horn delay  
	Uses Events and has 5 that can be uassigned that are location specific and a common events for the Actuator Extended/Retracted Time-out faults 

	Regardless of the travel of the actuator, the following define the extended and retracted positions
		Extended is the position expected when the solenoid valve is actuated
		Retracted is the position expected when the solenoid valve is resting
*)

VAR_IN_OUT
	CFG_EquipIndex				: DINT;	// Index used for local Equipment status array
	{attribute 'OPC.UA.DA' := '1'}
	Sts_EquipState					: ST_EquipmentStatus;		// State Status
END_VAR
VAR_INPUT
	{attribute 'OPC.UA.DA' := '1'}
	In_o_EquipStatePB				: ST_StateCntrlPB;		// Hmi push buttons to change states
	In_p_EquipStatePB				: ST_StateCntrlPB;		// programming to change states
	In_P_SVReqExtend			: BOOL;		// Input to extend actuator if in auto and conditions are met
	In_SimActive				: BOOL;
	In_EquipInit					: BOOL;		// Initialise;
	{attribute 'OPC.UA.DA' := '1'}
	In_EquipExtdFdbck			: BOOL := FALSE;	// Actuator Extended Feedback (1 = Extended)
	{attribute 'OPC.UA.DA' := '1'}
	In_EquipRtrcdFdbck			: BOOL := FALSE;	// Actuator Retracted Feedback (1 = Retracted)
	Cfg_EquipDefState				: E_StateCntrl;
	{attribute 'OPC.UA.DA' := '1'}
	Cfg_EquipLabel					: STRING(20);		// Label of the Solenoid
	Cfg_UseExtedFdbc			: BOOL := FALSE;	// Use Feedback from actuator for Extended state, otherwise, use output 

	// Events
	In_EquipEvents					: UINT;		// Event that is specific to the instance of the solenoid/actuator
	{attribute 'OPC.UA.DA' := '0'}
	Cfg_EquipEvntsArry				: ARRAY [0..15] OF ST_CfgEvents;
	Cfg_ExtendDetectTime		: TIME;
	Cfg_RetractDetectTime		: TIME;
	
	// Interlocks that can be Instance Specific
	In_EquipIntlks					: UINT;		// Interlock that is specific to the instance of the solenoid/actuator
	{attribute 'OPC.UA.DA' := '0'}
	Cfg_EquipIntlksArry			: ARRAY [0..15] OF ST_CfgEvents;		// Descriptions of the Interlock 
	
END_VAR
VAR_OUTPUT
	{attribute 'OPC.UA.DA' := '1'}
	Out_ExtendCrntSV			: BOOL;		// Extend command for the current solenoid/actuator
	{attribute 'OPC.UA.DA' := '1'}
	Sts_ExtendCrntSV			: BOOL;		// Status showing that current solenoid/actuator is extended/extending
	{attribute 'OPC.UA.DA' := '1'}
	Sts_All_Intlks_OK			: BOOL;		// Status bit to show that all interloks are good to Run 
	{attribute 'OPC.UA.DA' := '1'}
	Sts_FaultActive				: BOOL;	// Status Bit Showing that a fault is present (0= No Active Faults, 1= Fault Active)
	{attribute 'OPC.UA.DA' := '1'}
	Sts_WarnActive				: BOOL;	// Status Bit Showing that a warning is present (0= No Active Warnings, 1= Warning Active)
	{attribute 'OPC.UA.DA' := '1'}
	Sts_All_Evnts_OK			: BOOL;		// Status Bit Showing that ALL Events are OK to RUN (0= Event Present, 1= OK to Run)
	{attribute 'OPC.UA.DA' := '1'}
	Sts_IntlksArry				: ARRAY[0..15] OF ST_EventSts;		// Interlock status 0 to 15 Input
	{attribute 'OPC.UA.DA' := '1'}
	Sts_FaultsArry				: ARRAY[0..15] OF ST_EventSts;	// Status of each Fault Event State (0= OFF, 1=ON)
	{attribute 'OPC.UA.DA' := '1'}
	Sts_WarnsArry				: ARRAY[0..15] OF ST_EventSts;		// Status of each Warning Event State (0= OFF, 1=ON)
	{attribute 'OPC.UA.DA' := '0'}
	Sts_EvntsArry				: ARRAY[0..15] OF ST_EventSts; 	// Status of each Event State (0= OFF, 1=ON)
END_VAR
VAR
	{attribute 'OPC.UA.DA' := '0'}
	SV_fbIntrlks				: FB_Intlks_Latch;
	SV_IntlksArry				: ARRAY[0..15] OF BOOL;
	{attribute 'OPC.UA.DA' := '0'}
	SV_fbEquipCntrl				: FB_EquipCntrl;
	{attribute 'OPC.UA.DA' := '0'}
	SV_EventManager				: FB_EventMngr;
	SV_ExtendFault				: FB_JamDetect;			// This FB can also detect when it takes to long to extend an actuator
	SV_RetractFault				: FB_JamDetect;			// This FB can also detect when it takes to long to retract an actuator
	SV_EventArry				: ARRAY[0..15] OF BOOL;
	
	SV_LatchIgnore				: BOOL := FALSE;		// Put as a place holder for ease of future use
	SV_LatchReset				: BOOL := FALSE;		//Put as a place holder for ease of future use
	SV_IntlkBypassed			: ARRAY [0..15] OF BOOL;		//Put as a place holder for ease of future use
	SV_MoveEnabled				: BOOL;					// TRUE = Enable the SV/Actuator to operate
	SV_StartEnabled				: BOOL;					// TRUE = Start Motion for SV/actuator

END_VAR

// Set Up Common Single-Acting solenoid Interlocks and inputs for interlocks that are specific for the configuration instance
SV_IntlksArry[0] := In_EquipIntlks.0;
SV_IntlksArry[1] := System.SysIntlksAllOk; 
SV_IntlksArry[2] := In_EquipIntlks.2;
SV_IntlksArry[3] := In_EquipIntlks.3;
SV_IntlksArry[4] := In_EquipIntlks.4;
SV_IntlksArry[5] := In_EquipIntlks.5;
SV_IntlksArry[6] := In_EquipIntlks.6;
SV_IntlksArry[7] := In_EquipIntlks.7;
SV_IntlksArry[8] := In_EquipIntlks.8;
SV_IntlksArry[9] := In_EquipIntlks.9; 
SV_IntlksArry[10] := In_EquipIntlks.10;
SV_IntlksArry[11] := In_EquipIntlks.11;
SV_IntlksArry[12] := In_EquipIntlks.12;
SV_IntlksArry[13] := In_EquipIntlks.13;
SV_IntlksArry[14] := In_EquipIntlks.14;
SV_IntlksArry[15] := In_EquipIntlks.15;
	
// Call Interlock block
SV_fbIntrlks(
	In_Intlks:= SV_IntlksArry,
	CFG_IntlksArry:= Cfg_EquipIntlksArry, 
	HMI_LatchIgnore:= SV_LatchIgnore, 
	HMI_LatchReset:= SV_LatchReset, 
	All_Intlk_OK=> Sts_All_Intlks_OK, 
	STS_Intlks=> Sts_IntlksArry);
	
// Set Up Common Solenoid Events and inputs for events that are specific for the configuration instance
SV_EventArry[0]:= SV_ExtendFault.JamDetected;	// Even though this is a JamDetected output, it is really a Extend time-out fault
SV_EventArry[1]:= SV_RetractFault.JamDetected;	// Even though this is a JamDetected output, it is really a retract time-out fault
SV_EventArry[2]:= In_EquipEvents.2;
SV_EventArry[3]:= In_EquipEvents.3;
SV_EventArry[4]:= In_EquipEvents.4;
SV_EventArry[5]:= In_EquipEvents.5;
SV_EventArry[6]:= In_EquipEvents.6;
SV_EventArry[7]:= In_EquipEvents.7;
SV_EventArry[8]:= In_EquipEvents.8;
SV_EventArry[9]:= In_EquipEvents.9;
SV_EventArry[10]:= In_EquipEvents.10;
SV_EventArry[11]:= In_EquipEvents.11;
SV_EventArry[12]:= In_EquipEvents.12;
SV_EventArry[13]:= In_EquipEvents.13;
SV_EventArry[14]:= In_EquipEvents.14;
SV_EventArry[15]:= In_EquipEvents.15;

// Event Manager
SV_EventManager(
	sEquipStateCntrlSts := Sts_EquipState.Sts_EquipmentState,
	In_EventsArry := SV_EventArry ,  
	CFG_EvntsArry:= Cfg_EquipEvntsArry, 
	HMI_LatchReset:= In_o_EquipStatePB.ResetPB OR In_p_EquipStatePB.ResetPB,
	Out_FaultActive=> Sts_FaultActive, 
	Out_WarnActive=> Sts_WarnActive, 
	Sts_All_Evnts_OK=> Sts_All_Evnts_OK, 
	Sts_FaultsArry=> Sts_FaultsArry, 
	Sts_WarnsArry=> Sts_WarnsArry, 
	Sts_EvntsArry=> Sts_EvntsArry);
	
(*
	Set up individual Events that are common for this configuration
 	For the Extend Fault, use one of two conditions
		1 - If the SV is configured to use Extended feedback, check the input
		2 - If the SV is not configured to use Extedned feedback, check that the output is on and the retracted input is not on
*)
SV_ExtendFault.In_PE := (Cfg_UseExtedFdbc AND NOT In_EquipExtdFdbck) OR (NOT Cfg_UseExtedFdbc AND (Out_ExtendCrntSV AND In_EquipRtrcdFdbck));
SV_ExtendFault(
	In_Status:= Out_ExtendCrntSV, 
	CFG_PEOKState:= 0, 
	JamDetTime:= cfg_ExtendDetectTime);
	
(*
 	For the Retract Fault, use the following condition
		Output is off and the actuator is not in the retracted condition
*)
SV_RetractFault.In_PE := NOT Out_ExtendCrntSV AND NOT In_EquipRtrcdFdbck;
SV_RetractFault(
	In_Status:= NOT Out_ExtendCrntSV, 
	CFG_PEOKState:= 0, 
	JamDetTime:= cfg_RetractDetectTime);

//Call Equipment FB to control current SV/Actuator	
SV_fbEquipCntrl(
	CFG_EquipIndex := cfg_EquipIndex,
	CFG_EquipLabel := Cfg_EquipLabel,
	CFG_UseStrtCnd:= FALSE, 
	CFG_UseIntrlks:= TRUE, 
	CFG_UseHrnDly:= FALSE, 
	CFG_EquipDefState:= Cfg_EquipDefState, 
	In_IntlksOK:= Sts_All_Intlks_OK, 
	In_SimActive:= In_SimActive, 
	In_Init:= In_EquipInit, 
	o_EquipStatePB:= In_o_EquipStatePB, 
	p_EquipStatePB:= In_p_EquipStatePB, 
	P_EquipReqRun:= In_P_SVReqExtend, 
	In_EquipFaults:= Sts_FaultActive, 
	Out_EquipRun=> , 
	Out_Horn=> , 
	Sts_EquipState:= Sts_EquipState.Sts_EquipmentState);	

// Process the SV_MoveEnabled signal
SV_MoveEnabled := SV_fbEquipCntrl.Out_EquipRun;

SV_StartEnabled := SV_MoveEnabled;	

// Actuate the SV based on the results of the Equipment Control state
IF Sts_EquipState.Sts_EquipmentState.CrntState = E_StateCntrl.stAuto THEN
	IF (In_P_SVReqExtend )
	   THEN
		Out_ExtendCrntSV := SV_StartEnabled;
		// Set Solenoid Actuation Status
		Sts_ExtendCrntSV := (Out_ExtendCrntSV) OR (In_SimActive AND SV_fbEquipCntrl.RunApproved);
	ELSE
		Out_ExtendCrntSV := FALSE;
		// Set Solenoid Actuation Status
		Sts_ExtendCrntSV := FALSE;
	END_IF
ELSE
	IF (In_o_EquipStatePB.ManExtendPB)
	   THEN
		Out_ExtendCrntSV := SV_StartEnabled;
		// Set Solenoid Actuation Status
		Sts_ExtendCrntSV := (Out_ExtendCrntSV) OR (In_SimActive AND SV_fbEquipCntrl.RunApproved);
	ELSE
		Out_ExtendCrntSV := FALSE;
		// Set Solenoid Actuation Status
		Sts_ExtendCrntSV := FALSE;
	END_IF
END_IF

// Turn OFF Extend and Retract when a stop is issued
IF In_p_EquipStatePB.StopPB OR In_o_EquipStatePB.StopPB THEN
	Out_ExtendCrntSV := FALSE;
	Sts_ExtendCrntSV := FALSE;
END_IF

// Capture the Operation state of the Solenoid/actuator
IF Sts_ExtendCrntSV THEN
	// Solenoid Actuating/Entending
	Sts_EquipState.Sts_EquipmentState.CrntOperState := E_OperStateCntrl.extending;
	// Solenoid Extended
	IF (Cfg_UseExtedFdbc AND In_EquipExtdFdbck) OR (NOT Cfg_UseExtedFdbc AND (Out_ExtendCrntSV AND NOT In_EquipRtrcdFdbck)) THEN
		Sts_EquipState.Sts_EquipmentState.CrntOperState := E_OperStateCntrl.extended;
	END_IF
ELSE
	// Solenoid Retracting
	Sts_EquipState.Sts_EquipmentState.CrntOperState := E_OperStateCntrl.retracting;
	// Solenoid Retracted
	IF In_EquipRtrcdFdbck THEN
		Sts_EquipState.Sts_EquipmentState.CrntOperState := E_OperStateCntrl.retracted;
	END_IF
END_IF
IF NOT Sts_ExtendCrntSV
   AND NOT In_EquipRtrcdFdbck
   AND NOT (Cfg_UseExtedFdbc AND In_EquipExtdFdbck) OR (NOT Cfg_UseExtedFdbc AND (Out_ExtendCrntSV AND NOT In_EquipRtrcdFdbck)) 
   THEN
	Sts_EquipState.Sts_EquipmentState.CrntOperState := E_OperStateCntrl.unknown;
END_IF
// Solenoid control and state
CASE Sts_EquipState.Sts_EquipmentState.CrntOperState OF
	E_OperStateCntrl.extended:
			Sts_EquipState.Sts_IsExtended := TRUE;
			Sts_EquipState.Sts_IsExtending := FALSE;
			Sts_EquipState.Sts_IsRetracted := FALSE;
			Sts_EquipState.Sts_IsRetracting := FALSE;
	E_OperStateCntrl.extending:
			Sts_EquipState.Sts_IsExtended := FALSE;
			Sts_EquipState.Sts_IsExtending := TRUE;
			Sts_EquipState.Sts_IsRetracted := FALSE;
			Sts_EquipState.Sts_IsRetracting := FALSE;
	E_OperStateCntrl.retracted:
			Sts_EquipState.Sts_IsExtended := FALSE;
			Sts_EquipState.Sts_IsExtending := FALSE;
			Sts_EquipState.Sts_IsRetracted := TRUE;
			Sts_EquipState.Sts_IsRetracting := FALSE;
	E_OperStateCntrl.retracting:
			Sts_EquipState.Sts_IsExtended := FALSE;
			Sts_EquipState.Sts_IsExtending := FALSE;
			Sts_EquipState.Sts_IsRetracted := FALSE;
			Sts_EquipState.Sts_IsRetracting := TRUE;
END_CASE

// Populate the Sts Output Variables
Sts_EquipState.Sts_All_Intlks_OK  := Sts_All_Intlks_OK;
Sts_EquipState.Sts_All_Evnts_OK  := Sts_All_Evnts_OK;
Sts_EquipState.Sts_FaultActive := Sts_FaultActive;
Sts_EquipState.Sts_WarnActive := Sts_WarnActive;

END_FUNCTION_BLOCK

// ---- POUs/FunctionBlocks/Solenoids/Functions/FB_Solenoid_DA.TcPOU
FUNCTION_BLOCK FB_Solenoid_DA

(* Double-Acting solenoid Set up,
	Uses Interlocks. No common interlocks
	Doesn't use Start Conditions or the horn delay  
	Uses Events and has 5 that can be uassigned that are location specific and a common events for the Actuator Extended/Retracted Time-out faults 

	Regardless of the travel of the actuator, the following define the extended and retracted positions
		Extended is the position expected when the solenoid valve is actuated
		Retracted is the position expected when the solenoid valve is resting
*)

VAR_IN_OUT
	CFG_EquipIndex				: DINT;	// Index used for local Equipment status array
	{attribute 'OPC.UA.DA' := '1'}
	Sts_EquipState					: ST_EquipmentStatus;		// State Status
END_VAR
VAR_INPUT
	{attribute 'OPC.UA.DA' := '1'}
	In_o_EquipStatePB				: ST_StateCntrlPB;		// Hmi push buttons to change states
	In_p_EquipStatePB				: ST_StateCntrlPB;		// programming to change states
	In_P_SVReqExtend			: BOOL;		// Input to extend actuator if in auto and conditions are met
	In_P_SVReqRetract			: BOOL;		// Input to retract actuator if in auto and conditions are met
	In_SimActive				: BOOL;
	In_EquipInit					: BOOL;		// Initialise;
	{attribute 'OPC.UA.DA' := '1'}
	In_EquipExtdFdbck			: BOOL := FALSE;	// Actuator Extended Feedback (1 = Extended)
	{attribute 'OPC.UA.DA' := '1'}
	In_EquipRtrcdFdbck			: BOOL := FALSE;	// Actuator Retracted Feedback (1 = Retracted)
	Cfg_EquipDefState				: E_StateCntrl;
	{attribute 'OPC.UA.DA' := '1'}
	Cfg_EquipLabel					: STRING(20);		// Label of the Solenoid
	Cfg_UseExtedFdbc			: BOOL := FALSE;	// Use Feedback from actuator for Extended state, otherwise, use output 

	// Events
	// This is the system interlock, but could be something different
	In_EquipEvents					: UINT;		// Event that is specific to the instance of the solenoid/actuator
	{attribute 'OPC.UA.DA' := '0'}
	Cfg_EquipEvntsArry				: ARRAY [0..15] OF ST_CfgEvents;
	Cfg_ExtendDetectTime		: TIME;
	Cfg_RetractDetectTime		: TIME;
	
	// Interlocks that can be Instance Specific
	In_EquipIntlks					: UINT;		// Interlock that is specific to the instance of the solenoid/actuator
	{attribute 'OPC.UA.DA' := '0'}
	Cfg_EquipIntlksArry			: ARRAY [0..15] OF ST_CfgEvents;		// Descriptions of the Interlock 
	
END_VAR
VAR_OUTPUT
	{attribute 'OPC.UA.DA' := '1'}
	Out_ExtendCrntSV			: BOOL;		// Extend command for the current solenoid/actuator
	{attribute 'OPC.UA.DA' := '1'}
	Sts_ExtendCrntSV			: BOOL;		// Status showing that current solenoid/actuator is extended/extending
	{attribute 'OPC.UA.DA' := '1'}
	Out_RetractCrntSV			: BOOL;		// Retract command for the current solenoid/actuator
	{attribute 'OPC.UA.DA' := '1'}
	Sts_RetractCrntSV			: BOOL;		// Status showing that current solenoid/actuator is retracteded/retractinging
	{attribute 'OPC.UA.DA' := '1'}
	Sts_All_Intlks_OK			: BOOL;		// Status bit to show that all interloks are good to Run 
	{attribute 'OPC.UA.DA' := '1'}
	Sts_FaultActive				: BOOL;	// Status Bit Showing that a fault is present (0= No Active Faults, 1= Fault Active)
	{attribute 'OPC.UA.DA' := '1'}
	Sts_WarnActive				: BOOL;	// Status Bit Showing that a warning is present (0= No Active Warnings, 1= Warning Active)
	{attribute 'OPC.UA.DA' := '1'}
	Sts_All_Evnts_OK			: BOOL;		// Status Bit Showing that ALL Events are OK to RUN (0= Event Present, 1= OK to Run)
	{attribute 'OPC.UA.DA' := '1'}
	Sts_IntlksArry				: ARRAY[0..15] OF ST_EventSts;		// Interlock status 0 to 15 Input
	{attribute 'OPC.UA.DA' := '1'}
	Sts_FaultsArry				: ARRAY[0..15] OF ST_EventSts;	// Status of each Fault Event State (0= OFF, 1=ON)
	{attribute 'OPC.UA.DA' := '1'}
	Sts_WarnsArry				: ARRAY[0..15] OF ST_EventSts;		// Status of each Warning Event State (0= OFF, 1=ON)
	{attribute 'OPC.UA.DA' := '0'}
	Sts_EvntsArry				: ARRAY[0..15] OF ST_EventSts; 	// Status of each Event State (0= OFF, 1=ON)
END_VAR
VAR
	{attribute 'OPC.UA.DA' := '0'}
	SV_fbIntrlks				: FB_Intlks_Latch;
	SV_IntlksArry				: ARRAY[0..15] OF BOOL;
	{attribute 'OPC.UA.DA' := '0'}
	SV_fbEquipCntrl				: FB_EquipCntrl;
	{attribute 'OPC.UA.DA' := '0'}
	SV_EventManager				: FB_EventMngr;
	SV_ExtendFault				: FB_JamDetect;			// This FB can also detect when it takes to long to extend an actuator
	SV_RetractFault				: FB_JamDetect;			// This FB can also detect when it takes to long to retract an actuator
	SV_EventArry				: ARRAY[0..15] OF BOOL;
	
	SV_LatchIgnore				: BOOL := FALSE;		// Put as a place holder for ease of future use
	SV_LatchReset				: BOOL := FALSE;		//Put as a place holder for ease of future use
	SV_IntlkBypassed			: ARRAY [0..15] OF BOOL;		//Put as a place holder for ease of future use
	SV_MoveEnabled				: BOOL;					// TRUE = Enable the SV/Actuator to operate
	SV_StartEnabled				: BOOL;					// TRUE = Start Motion for SV/actuator

END_VAR

// Set Up Common Single-Acting solenoid Interlocks and inputs for interlocks that are specific for the configuration instance
SV_IntlksArry[0] := In_EquipIntlks.0;
SV_IntlksArry[1] := System.SysIntlksAllOk; 
SV_IntlksArry[2] := In_EquipIntlks.2;
SV_IntlksArry[3] := In_EquipIntlks.3;
SV_IntlksArry[4] := In_EquipIntlks.4;
SV_IntlksArry[5] := In_EquipIntlks.5;
SV_IntlksArry[6] := In_EquipIntlks.6;
SV_IntlksArry[7] := In_EquipIntlks.7;
SV_IntlksArry[8] := In_EquipIntlks.8;
SV_IntlksArry[9] := In_EquipIntlks.9; 
SV_IntlksArry[10] := In_EquipIntlks.10;
SV_IntlksArry[11] := In_EquipIntlks.11;
SV_IntlksArry[12] := In_EquipIntlks.12;
SV_IntlksArry[13] := In_EquipIntlks.13;
SV_IntlksArry[14] := In_EquipIntlks.14;
SV_IntlksArry[15] := In_EquipIntlks.15;
	
// Call Interlock block
SV_fbIntrlks(
	In_Intlks:= SV_IntlksArry,
	CFG_IntlksArry:= Cfg_EquipIntlksArry, 
	HMI_LatchIgnore:= SV_LatchIgnore, 
	HMI_LatchReset:= SV_LatchReset, 
	All_Intlk_OK=> Sts_All_Intlks_OK, 
	STS_Intlks=> Sts_IntlksArry);
	
// Set Up Common Solenoid Events and inputs for events that are specific for the configuration instance
SV_EventArry[0]:= SV_ExtendFault.JamDetected;	// Even though this is a JamDetected output, it is really a Extend time-out fault
SV_EventArry[1]:= SV_RetractFault.JamDetected;	// Even though this is a JamDetected output, it is really a retract time-out fault
SV_EventArry[2]:= In_EquipEvents.2;
SV_EventArry[3]:= In_EquipEvents.3;
SV_EventArry[4]:= In_EquipEvents.4;
SV_EventArry[5]:= In_EquipEvents.5;
SV_EventArry[6]:= In_EquipEvents.6;
SV_EventArry[7]:= In_EquipEvents.7;
SV_EventArry[8]:= In_EquipEvents.8;
SV_EventArry[9]:= In_EquipEvents.9;
SV_EventArry[10]:= In_EquipEvents.10;
SV_EventArry[11]:= In_EquipEvents.11;
SV_EventArry[12]:= In_EquipEvents.12;
SV_EventArry[13]:= In_EquipEvents.13;
SV_EventArry[14]:= In_EquipEvents.14;
SV_EventArry[15]:= In_EquipEvents.15;

// Event Manager
SV_EventManager(
	sEquipStateCntrlSts := Sts_EquipState.Sts_EquipmentState,
	In_EventsArry := SV_EventArry ,  
	CFG_EvntsArry:= Cfg_EquipEvntsArry, 
	HMI_LatchReset:= In_o_EquipStatePB.ResetPB OR In_p_EquipStatePB.ResetPB,
	Out_FaultActive=> Sts_FaultActive, 
	Out_WarnActive=> Sts_WarnActive, 
	Sts_All_Evnts_OK=> Sts_All_Evnts_OK, 
	Sts_FaultsArry=> Sts_FaultsArry, 
	Sts_WarnsArry=> Sts_WarnsArry, 
	Sts_EvntsArry=> Sts_EvntsArry);
	
(*
	Set up individual Events that are common for this configuration
 	For the Extend Fault, use one of two conditions
		1 - If the SV is configured to use Extended feedback, check the input
		2 - If the SV is not configured to use Extedned feedback, check that the output is on and the retracted input is not on
*)
SV_ExtendFault.In_PE := (Cfg_UseExtedFdbc AND NOT In_EquipExtdFdbck) OR (NOT Cfg_UseExtedFdbc AND (Out_ExtendCrntSV AND In_EquipRtrcdFdbck));
SV_ExtendFault(
	In_Status:= NOT In_o_EquipStatePB.ResetPB AND Out_ExtendCrntSV, 
	CFG_PEOKState:= 0, 
	JamDetTime:= cfg_ExtendDetectTime);
	
(*
 	For the Retract Fault, use the following condition
		Retracted Output is ON and the actuator is not in the retracted condition
*)
SV_RetractFault.In_PE := Out_RetractCrntSV AND NOT In_EquipRtrcdFdbck;
SV_RetractFault(
	In_Status:= NOT In_o_EquipStatePB.ResetPB AND Out_RetractCrntSV, 
	CFG_PEOKState:= 0, 
	JamDetTime:= cfg_RetractDetectTime);

//Call Equipment FB to control current SV/Actuator	
// XOR the Extend and Retract. The interlocks/events must be prefixed with the extend or retract command 
SV_fbEquipCntrl(
	CFG_EquipIndex := cfg_EquipIndex,
	CFG_EquipLabel := Cfg_EquipLabel,
	CFG_UseStrtCnd:= FALSE, 
	CFG_UseIntrlks:= TRUE, 
	CFG_UseHrnDly:= FALSE, 
	CFG_EquipDefState:= Cfg_EquipDefState, 
	In_IntlksOK:= Sts_All_Intlks_OK, 
	In_SimActive:= In_SimActive, 
	In_Init:= In_EquipInit, 
	o_EquipStatePB:= In_o_EquipStatePB, 
	p_EquipStatePB:= In_p_EquipStatePB, 
	P_EquipReqRun:= In_P_SVReqExtend XOR In_P_SVReqRetract, 
	In_EquipFaults:= Sts_FaultActive, 
	Out_EquipRun=> , 
	Out_Horn=> , 
	Sts_EquipState:= Sts_EquipState.Sts_EquipmentState);	

// Process the SV_MoveEnabled signal
SV_MoveEnabled := SV_fbEquipCntrl.Out_EquipRun;

SV_StartEnabled := SV_MoveEnabled;	

// Actuate the SV based on the results of the Equipment Control state
IF Sts_EquipState.Sts_EquipmentState.CrntState = E_StateCntrl.stAuto THEN
	IF (In_P_SVReqExtend AND NOT In_P_SVReqRetract)
	   THEN
		Out_RetractCrntSV := FALSE;
		Out_ExtendCrntSV := SV_StartEnabled;
		// Set Solenoid Actuation Status
		Sts_ExtendCrntSV := (Out_ExtendCrntSV) OR (In_SimActive AND SV_fbEquipCntrl.RunApproved);
		Sts_RetractCrntSV := FALSE;
	END_IF
	IF In_P_SVReqRetract THEN
		Out_RetractCrntSV := SV_StartEnabled;
		Out_ExtendCrntSV := FALSE;
		// Set Solenoid Actuation Status
		Sts_RetractCrntSV := (Out_RetractCrntSV) OR (In_SimActive AND SV_fbEquipCntrl.RunApproved);
		Sts_ExtendCrntSV := FALSE;
	END_IF
ELSE
	IF (In_o_EquipStatePB.ManExtendPB AND NOT In_o_EquipStatePB.ManRetractPB)
	   THEN
		Out_RetractCrntSV := FALSE;
		Out_ExtendCrntSV := SV_StartEnabled;
		// Set Solenoid Actuation Status
		Sts_ExtendCrntSV := (Out_ExtendCrntSV) OR (In_SimActive AND SV_fbEquipCntrl.RunApproved);
		Sts_RetractCrntSV := FALSE;
	END_IF
	IF In_o_EquipStatePB.ManRetractPB THEN
		Out_RetractCrntSV := SV_StartEnabled;
		Out_ExtendCrntSV := FALSE;
		// Set Solenoid Actuation Status
		Sts_RetractCrntSV := (Out_RetractCrntSV) OR (In_SimActive AND SV_fbEquipCntrl.RunApproved);
		Sts_ExtendCrntSV := FALSE;
	END_IF
END_IF

// Turn OFF Extend and Retract when a stop is issued
IF In_p_EquipStatePB.StopPB OR In_o_EquipStatePB.StopPB THEN
	Out_ExtendCrntSV := FALSE;
	Out_RetractCrntSV := FALSE;
	Sts_ExtendCrntSV := FALSE;
	Sts_RetractCrntSV := FALSE;
END_IF

// Capture the Operation state of the Solenoid/actuator
IF Sts_ExtendCrntSV THEN
	// Solenoid Actuating/Entending
	Sts_EquipState.Sts_EquipmentState.CrntOperState := E_OperStateCntrl.extending;
	// Solenoid Extended
	IF (Cfg_UseExtedFdbc AND In_EquipExtdFdbck) OR (NOT Cfg_UseExtedFdbc AND (Out_ExtendCrntSV AND NOT In_EquipRtrcdFdbck)) THEN
		Sts_EquipState.Sts_EquipmentState.CrntOperState := E_OperStateCntrl.extended;
	END_IF
END_IF
IF Sts_RetractCrntSV THEN
	// Solenoid Retracting
	Sts_EquipState.Sts_EquipmentState.CrntOperState := E_OperStateCntrl.retracting;
	// Solenoid Retracted
	IF In_EquipRtrcdFdbck THEN
		Sts_EquipState.Sts_EquipmentState.CrntOperState := E_OperStateCntrl.retracted;
	END_IF
END_IF
IF NOT Sts_ExtendCrntSV
   AND NOT Sts_RetractCrntSV 
   AND NOT In_EquipRtrcdFdbck
   AND NOT (Cfg_UseExtedFdbc AND In_EquipExtdFdbck) OR (NOT Cfg_UseExtedFdbc AND (Out_ExtendCrntSV AND NOT In_EquipRtrcdFdbck)) 
   THEN
	Sts_EquipState.Sts_EquipmentState.CrntOperState := E_OperStateCntrl.unknown;
END_IF
// Solenoid control and state
CASE Sts_EquipState.Sts_EquipmentState.CrntOperState OF
	E_OperStateCntrl.extended:
			Sts_EquipState.Sts_IsExtended := TRUE;
			Sts_EquipState.Sts_IsExtending := FALSE;
			Sts_EquipState.Sts_IsRetracted := FALSE;
			Sts_EquipState.Sts_IsRetracting := FALSE;
	E_OperStateCntrl.extending:
			Sts_EquipState.Sts_IsExtended := FALSE;
			Sts_EquipState.Sts_IsExtending := TRUE;
			Sts_EquipState.Sts_IsRetracted := FALSE;
			Sts_EquipState.Sts_IsRetracting := FALSE;
	E_OperStateCntrl.retracted:
			Sts_EquipState.Sts_IsExtended := FALSE;
			Sts_EquipState.Sts_IsExtending := FALSE;
			Sts_EquipState.Sts_IsRetracted := TRUE;
			Sts_EquipState.Sts_IsRetracting := FALSE;
	E_OperStateCntrl.retracting:
			Sts_EquipState.Sts_IsExtended := FALSE;
			Sts_EquipState.Sts_IsExtending := FALSE;
			Sts_EquipState.Sts_IsRetracted := FALSE;
			Sts_EquipState.Sts_IsRetracting := TRUE;
END_CASE

// Populate the Sts Output Variables
Sts_EquipState.Sts_All_Intlks_OK  := Sts_All_Intlks_OK;
Sts_EquipState.Sts_All_Evnts_OK  := Sts_All_Evnts_OK;
Sts_EquipState.Sts_FaultActive := Sts_FaultActive;
Sts_EquipState.Sts_WarnActive := Sts_WarnActive;

END_FUNCTION_BLOCK

// ---- POUs/Singulation_Control.TcPOU
PROGRAM Singulation_Control
VAR
	SortSingulation	:	FB_Singulation;
	RetryLimit		:	UINT := 1;
	ReleaseDist		:	UINT;
END_VAR

SortSingulation(
In_ConveyorRunning := Conveyors.P6040_Status.Sts_IsRunning,
	In_Grabber_1_Auto := Solenoids.GR6040_01_Status.Sts_EquipmentState.StsAuto,
 	In_Grabber_1_Extended := ProxSensors.In_PX_6261_Extended,
	In_Grabber_1_Retracted := ProxSensors.In_PX_6241_Retracted,
	In_Grabber_2_Auto := Solenoids.GR6040_02_Status.Sts_EquipmentState.StsAuto,
	In_Grabber_2_Extended := ProxSensors.In_PX_6151_Extended,
	In_Grabber_2_Retracted := ProxSensors.In_PX_6121_Retracted,
	In_PinStop_Auto := Solenoids.PI6040_01_Status.Sts_EquipmentState.StsAuto,
	In_PinStop_Extended := ProxSensors.In_PX_6152_Extended,
	In_PinStop_Retracted := ProxSensors.In_PX_6122_Retracted,
	In_FaultReset := System.Cnvyr_Reset,
	In_EncoderCount := GVL_IO.ENC_9021_Raw,
	In_PE_GrabTrigger:= PhotoEyes.PE_6201.Out_OnFltrd, 
	In_PE_ToteTrigger:= PhotoEyes.PE_6181.Out_OffFltrd, 
	In_PE_ClearedTrigger:= PhotoEyes.PE_6241.Out_OffFltrd,
	Cfg_GappingDistance := ReleaseDist,
	Cfg_TimeOutTime:= T#5S,
	Cfg_RetryLimit:= RetryLimit, 
);

END_PROGRAM

// ---- POUs/Sorter.TcPOU
PROGRAM Sorter
VAR
	nSorterClearIdx				: DINT;
	bSimulate					: BOOL := FALSE;	// Indicates when runing a simulation
	
	st_ToInduct					: ST_ItemTemporary;	// This is the next item to be inducted onto the sorter
	st_Inducting				: ST_ItemTemporary;	// This is the next item to be inducted onto the sorter
	st_InductUpdate				: ST_ItemTemporary;	// This is to update an item already being inducted
	{attribute 'OPC.UA.DA' := '1'}
	st_Sorter					: ST_Sorter;
	{attribute 'OPC.UA.DA' := '1'}
	aSorterDiverts 				: ARRAY[DIVERTMIN..NUMBEROFDIVERTS] OF ST_Divert;

	st_SorterEncoder 			: ST_Encoder;
	fb_SorterEncoder 			: FB_ProcessEncoder;


	tEncoderOK			: TON;
	nLastEncoderCount	: UDINT;

	{attribute 'OPC.UA.DA' := '1'}
	fb_SortMetrics				: FB_Metrics;

	In_DefaultDestination AT %I*	: DINT;	// Input default destination update from Host messaging(MsgControl.RECEIVE)

	fb_CommissionSorterDiverts	: FB_DivertCommission;
	rInductPE					: R_TRIG; 	// Capture the Rising edge of the Induct PE
	fInductPE					: F_TRIG; 	// Capture the Falling edge of the Induct PE

	rDischargePE				: R_TRIG; 	// Capture the Rising edge of the Discharge PE
	fDischargePE				: F_TRIG; 	// Capture the Falling edge of the Discharge PE

	st_TempItem					: ST_ItemTemporary;	// Store temporary Item info until BCR data is received

	DivertToCommission			: UINT := 0;	// Non-zero value will send all items to this divert

	sMessage			: STRING;

	ClearSorterArray	: BOOL;

	FB_DivertLog		: FB_DivertLog;
	FB_SorterLog		: FB_SorterLog;
	
	SorterDischargeItem	: ST_Item;
	
END_VAR

VAR PERSISTENT
	aSorterItems 				: ARRAY[SORTERENCODERMIN..SORTERENCODERMAX] OF ST_Item;	// Persist the Items to Sort array
	{attribute 'OPC.UA.DA' := '1'}
	st_SorterCfg				: ST_SorterConfig; 	// Persist Sorter configuration
	{attribute 'OPC.UA.DA' := '1'}
	aSorterDivertsCfgs 			: ARRAY[DIVERTMIN..NUMBEROFDIVERTS] OF ST_DivertCfg; 	// Persist Sorter Configuration
END_VAR

VAR CONSTANT
	SORTERMASKSIZE				: UINT := 12;		// Number of bits to mask into the Encoder Count, will define the size of the SORTERENCODERMAX value
	{attribute 'OPC.UA.DA' := '1'}
	NUMBEROFDIVERTS				: DINT := 5;
	DIVERTMIN					: DINT := 1;
	{attribute 'OPC.UA.DA' := '1'}
	SORTERENCODERMAX			: UDINT := ((LREAL_TO_UDINT(EXPT(2,SORTERMASKSIZE)))-1); // Calculated size based on the bitmask 
	{attribute 'OPC.UA.DA' := '1'}
	SORTERENCODERMIN			: UDINT := 0;

END_VAR

// Sorter clear when the system is restarted or downloaded (INIT=TRUE for first scan)
IF (GVL_IO.INIT AND NOT st_SorterCfg.RetainOnRestart) OR ClearSorterArray THEN
	FOR nSorterClearIdx := UDINT_TO_DINT(SORTERENCODERMIN) TO UDINT_TO_DINT(SORTERENCODERMAX) BY 1 DO
		IF nSorterLogEnable.SORTER_DUMP THEN
			IF aSorterItems[nSorterClearIdx].ID <> '' THEN
				IF .nSorterLogEnable.SORTER_DUMP THEN
					sMessage := CONCAT(' Item: ', aSorterItems[nSorterClearIdx].ID);
					sMessage := CONCAT(sMessage,' Index: ');
					sMessage := CONCAT(sMessage, DINT_TO_STRING(nSorterClearIdx));
					// Write to the Error List
					ADSLOGSTR( msgCtrlMask := ADSLOG_MSGTYPE_HINT OR ADSLOG_MSGTYPE_LOG
						, msgFmtStr := 'Array Dump Info: %s'
						, strArg := sMessage);
				END_IF
			END_IF
		END_IF
		aSorterItems[nSorterClearIdx] := BlankItem;
	END_FOR
	ClearSorterArray := FALSE;
END_IF

// Setup and process the Sorter Encoder
st_SorterEncoder.EncoderRawCount := GVL_IO.ENC_9021_Raw;
st_SorterEncoder.BitMaskSize := SORTERMASKSIZE;
fb_SorterEncoder(Encoder := st_SorterEncoder, Simulate := bSimulate);

(*
	Initializes the Diverts.  
*)
//Divert #1
aSorterDiverts[1].Config := aSorterDivertsCfgs[1];
aSorterDiverts[1].ConfirmPE := Photoeyes.PE_7191.Out; 			
aSorterDiverts[1].FullPE := Photoeyes.PE_7191.Out;   			

//Divert #2
aSorterDiverts[2].Config := aSorterDivertsCfgs[2];
aSorterDiverts[2].ConfirmPE := Photoeyes.PE_7241.Out; 		
aSorterDiverts[2].FullPE := Photoeyes.PE_7241.Out;   		

//Divert #3 
aSorterDiverts[3].Config := aSorterDivertsCfgs[3];
aSorterDiverts[3].ConfirmPE := Photoeyes.PE_8171.Out; 		
aSorterDiverts[3].FullPE := Photoeyes.PE_8171.Out;   	

//Divert #4 
aSorterDiverts[4].Config := aSorterDivertsCfgs[4];
aSorterDiverts[4].ConfirmPE := Photoeyes.PE_8221.Out; 		
aSorterDiverts[4].FullPE := Photoeyes.PE_8221.Out; 

//Divert #5
aSorterDiverts[5].Config := aSorterDivertsCfgs[5];
aSorterDiverts[5].ConfirmPE := Photoeyes.PE_8211.Out; 		
aSorterDiverts[5].FullPE := Photoeyes.PE_8211.Out; 	


fb_CommissionSorterDiverts(
			InductTrigger := Photoeyes.PE_7171.Out,
			ReferenceValue := st_SorterEncoder.CurrentCount, 
			DischargeTrigger := Photoeyes.PE_8211.Out,
			TestTime := T#10S, Diverts := aSorterDiverts);

// Provide a "hard-coded" default destination.
IF st_SorterCfg.DefaultDestination <= 0 THEN
	st_SorterCfg.DefaultDestination := 5;
END_IF						

// Name of the sorter equipment
st_SorterCfg.Name := Conveyors.cfgP6040Label;
st_SorterCfg.DivertCount := NUMBEROFDIVERTS;
IF DivertToCommission > 0 THEN
	st_SorterCfg.DefaultDestination := DivertToCommission;
END_IF
st_Sorter.EncoderCounts := st_SorterEncoder.CurrentCount;
st_Sorter.InductPE := PhotoEyes.PE_7171.Out;
st_Sorter.DischargePE := Photoeyes.PE_8211.Out;

// Test the Encoder
tEncoderOK.IN := (Conveyors.P6040_Status.Sts_IsRunning AND (st_Sorter.EncoderCounts = nLastEncoderCount));
nLastEncoderCount := st_Sorter.EncoderCounts;
tEncoderOK(PT:=T#1S);

// OK when Q is not on, but the alarm is reversed
  GVL_IO.ENC_9021_OK := tEncoderOK.Q;

// Publish the sorter name
  GVL_IO.SorterName := st_SorterCfg.Name;

  
  IF GVL_SorterItems.P6040_DefaultDestination <> st_SorterCfg.DefaultDestination THEN
	   st_SorterCfg.DefaultDestination := GVL_SorterItems.P6040_DefaultDestination; 
  END_IF
  
  
// Sorter
(*
	ProcessBuffers processes all associated buffers (Sorter/Divert/Arrival/Transport/Update)
	Items arriving at the sorter are detected and processed in this function block then deliverd to the SorterProgram
	Items inducted into sorter produce TransportResponse messages in this function block
	Items diverted off the sorter produce TransportComplete messages in this function block
*)
ProcessBuffers(st_NextToInduct := st_ToInduct
				, st_TempInductItem := st_TempItem
				, st_UpdateItem := st_Inducting
				, st_Sorter := st_Sorter
				, aDiverts := aSorterDiverts
				, aItems := aSorterItems
				, DivertToCommission := DivertToCommission
				, ItemsArrayMax := SORTERENCODERMAX
				, ItemsArrayMin := SORTERENCODERMIN
				,DefaultDestIdx => st_SorterCfg.DefaultDestIdx
				,RecircDestIdx => st_SorterCfg.RecircDestIdx);

// Sorter log logs induct/discharge PE's and prepares the Temporory Record for unidentified items
FB_SorterLog(
				SorterToLog := st_Sorter,
				SorterLogEnable := .nSorterLogEnable,
				ToInduct := st_ToInduct,
				TempItem => st_TempItem);

				
				
				
				
				
(*
	SorterProgram is a separate Program
	Config portion of the st_sorter is separate to allow it be be persistent.
*)
st_sorter.Config := st_sorterCfg;
Sorter_P6040(st_Sorter := st_Sorter
		, In_ItemToInduct := st_ToInduct.Item
		, In_InductingItem := st_Inducting.Item
		, aItems := aSorterItems
		, aDiverts := aSorterDiverts
		, st_tempItem := st_TempItem
		, ItemsArrayMax := SORTERENCODERMAX
		, ItemsArrayMin := SORTERENCODERMIN
		, DivertArrayMax := NUMBEROFDIVERTS
		, DivertArrayMin := DIVERTMIN
		, st_DischargeItem => SorterDischargeItem); 
//--------------------------------------Divert Config------------------------------------------
(*
	Initialize Diverts here. 
	Tie variables commented IO to physical IO address
*)

// LOG the diverts
FB_DivertLog(DivertArray := aSorterDiverts,
				DivertLogEnable := .nDivertLogEnable,
				EncoderCounts := st_SorterEncoder.CurrentCount);

END_PROGRAM

// ---- POUs/FunctionBlocks/Divert/Functions/FB_DivertCommission.TcPOU
FUNCTION_BLOCK FB_DivertCommission
VAR_INPUT
	InductTrigger	: BOOL; //This is the starting point you want to measure from
	ReferenceValue 	: UDINT; //This is the measurement reference you want to use (most typically will be an encoder value)
	DischargeTrigger: BOOL; //This is the end point that you want to stop measuring
	Reset			: BOOL; //1 - reset all values 0 - keep existing values
	TestTime 		: TIME; //Maximum amount of time it could possibly take to get measurement. If you're not getting a measurement, increase this time
END_VAR

VAR_IN_OUT
	Diverts			: ARRAY[*] OF ST_Divert; //Diverts that you want to measure
END_VAR

VAR
	DivertIndex		: DINT;
	StartCount 		: UDINT;
	EndCount 		: UDINT;
	InductFlag		: BOOL;
	NumberofDiverts	: DINT; 
	DivertLength 	: ARRAY[0..10] OF UDINT;
	DivertTime 		: ARRAY[0..10] OF TIME;
	DischargeFlag	: ARRAY[0..10] OF BOOL;
	
	DivertTimer 	: TON := (PT := TestTime);	
END_VAR

DivertTimer();

NumberofDiverts	:= UPPER_BOUND(Diverts,1);

IF NumberofDiverts < 10 THEN
	IF InductTrigger AND NOT InductFlag THEN
		StartCount := ReferenceValue;
		DivertTimer(IN := TRUE);
		InductFlag := TRUE;
	END_IF
	
	IF DischargeTrigger AND NOT DischargeFlag[0] THEN
		DivertLength[0] := ReferenceValue;
		DivertTime[0]   := DivertTimer.ET;
		DivertTimer(IN := FALSE);
		DischargeFlag[0] := TRUE;
	END_IF
	
	FOR DivertIndex := 1 TO NumberOfDiverts DO
		IF Diverts[DivertIndex].ConfirmPE AND NOT DischargeFlag[DivertIndex] THEN
			DivertLength[DivertIndex]  := ReferenceValue;
			DivertTime[DivertIndex]    := DivertTimer.ET;
			DischargeFlag[DivertIndex] := TRUE;	
		END_IF
	END_FOR
	
	IF Reset THEN
		InductFlag := FALSE;
		DivertTimer(IN := FALSE);
		FOR DivertIndex := 0 TO NumberOfDiverts DO
			DischargeFlag[DivertIndex] := FALSE;
			DivertLength[DivertIndex] := 0;
		END_FOR
	END_IF
END_IF

END_FUNCTION_BLOCK

// ---- POUs/FunctionBlocks/Sorter/Functions/FB_SorterLog.TcPOU
FUNCTION_BLOCK FB_SorterLog
VAR_IN_OUT
END_VAR
VAR_INPUT
	SorterToLog			:	ST_Sorter;
	SorterLogEnable		:	UDINT;
	ToInduct			:	ST_ItemTemporary;
END_VAR
VAR_OUTPUT
	TempItem			:	ST_ItemTemporary;
END_VAR
VAR
	rInductPE			:	R_TRIG;
	fInductPE			:	F_TRIG;
	rDischargePE		:	R_TRIG;
	fDischargePE		:	F_TRIG;
	sMessage			:	STRING;
	BlankItem			: 	ST_Item := (ID := ''
										, UniqueID := 0
										, Destination := 0
										, Status := E_StatusCode.No_Status
										, ExtStatus := E_StatusCode.No_Status
										, DeviceID := ''
										, MessageType := E_MessageIds.NoMessage_00);
END_VAR

// Capture rising and falling edge Triggers of the configured Sorter PE (Induct/Discharge)
rInductPE(CLK:= SorterToLog.InductPE, Q =>);
fInductPE(CLK:= SorterToLog.InductPE, Q =>);
rDischargePE(CLK:= SorterToLog.DischargePE, Q =>);
fDischargePE(CLK:= SorterToLog.DischargePE, Q =>);

// On the rising/falling edge of the Induct PE
IF rInductPE.Q OR fInductPE.Q THEN
	IF SorterLogEnable.SORTER_DISCHARGE_PE THEN
		// Write to the Error List
		ADSLOGSTR( msgCtrlMask := ADSLOG_MSGTYPE_HINT OR ADSLOG_MSGTYPE_LOG
			, msgFmtStr := 'Induct PE Blocked : %s'
			, strArg := BOOL_TO_STRING(SorterToLog.DischargePE)); 
	END_IF
END_IF

// Prepare a dummy record for items that arrive before BCR data is received
// On the rising edge of the Induct PE
IF rInductPE.Q THEN
	// Test for a UniqueID, which indicates that a Barcode has been received
	IF ToInduct.Item.UniqueID = 0 THEN
		// Capture and create relevant info
		TempItem.Counts := SorterToLog.EncoderCounts;
		TempItem.Item.UniqueID :=  UDINT_TO_DINT(SorterToLog.EncoderCounts);
		TempItem.Item.ID :=  CONCAT('T-', UDINT_TO_STRING(SorterToLog.EncoderCounts));
		TempItem.Item.Destination := SorterToLog.Config.DefaultDestination;
		TempItem.Item.Status := E_StatusCode.UnidentifiedItem;
		IF SorterLogEnable.SORTER_TEMPID THEN
			ADSLOGSTR( msgCtrlMask := ADSLOG_MSGTYPE_HINT OR ADSLOG_MSGTYPE_LOG
				, msgFmtStr := 'Temp ID Assigned : %s'
				, strArg := TempItem.Item.ID);
		END_IF
	END_IF	
END_IF

// Clear the dummy record when the PE clears
// Items can only be inducted when the BCR info is received before or while the induct PE is blocked
IF fInductPE.Q THEN
	// Clear the record
	TempItem.Counts := 0;
	TempItem.Item :=  BlankItem;
END_IF

// On the rising/falling edge of the Discharge PE
IF rDischargePE.Q OR fDischargePE.Q THEN
	IF SorterLogEnable.SORTER_DISCHARGE_PE THEN
		// Write to the Error List
		ADSLOGSTR( msgCtrlMask := ADSLOG_MSGTYPE_HINT OR ADSLOG_MSGTYPE_LOG
			, msgFmtStr := 'Discharge PE Blocked : %s'
			, strArg := BOOL_TO_STRING(SorterToLog.DischargePE)); 
	END_IF
END_IF

END_FUNCTION_BLOCK

// ---- POUs/FunctionBlocks/Sorter/ProcessBuffers.TcPOU
PROGRAM ProcessBuffers
VAR_IN_OUT
	st_NextToInduct					: ST_ItemTemporary;
	st_UpdateItem					: ST_ItemTemporary;
	st_TempInductItem				: ST_ItemTemporary;
	st_Sorter						: ST_Sorter;
	aDiverts						: ARRAY[SorterExample.DIVERTMIN..SorterExample.NUMBEROFDIVERTS] OF ST_DIVERT;
	aItems 							: ARRAY[SorterExample.SORTERENCODERMIN..SorterExample.SORTERENCODERMAX] OF ST_Item;
END_VAR

VAR_INPUT
	DivertToCommission				: DINT;
	ItemsArrayMax 					: UDINT;
	ItemsArrayMin 					: UDINT;
END_VAR
VAR
	st_ArrivalBuffer AT %I* 		: ST_ItemBuffer;
	st_ArrivalFdbkIn				: ST_ItemBufferFdbk;
	st_ArrivalFdbkOut	AT %Q*		: ST_ItemBufferFdbk;
	fb_ArrivalBuffer				: FB_ItemBuffer;
	st_ArrivalItem 					: ST_Item;		// Arrival Item (Bar code read) from System PLC (BarCodeReaders.pou)

	// Item to replace in the sorter buffer
	st_ReplaceItem					: st_Item;

	st_TransportBuffer AT %I* 		: ST_ItemBuffer;
	st_TransportFdbkIn				: ST_ItemBufferFdbk;
	st_TransportFdbkOut	AT %Q*		: ST_ItemBufferFdbk;
	fb_TransportBuffer				: FB_ItemBuffer;

	st_UpdateBuffer AT %Q* 			: ST_ItemBuffer;
	st_UpdateFdbkIn	AT %I*			: ST_ItemBufferFdbk;
	st_UpdateFdbkOut				: ST_ItemBufferFdbk;
	fb_UpdateBuffer 				: FB_ItemBuffer;

	st_ToUpdate						: ST_ItemTemporary;	// Item to Update on the Sorter, or waiting to be added to the sorter

	ItemsArraySize			: UDINT;

	TransportItemInSorter	: ST_Item;	// Temporary Processing Item
	TransportItemFound		: ST_Item;	// Item to Update Found
	TransportSorterIndex	: UDINT;

	ExitSorterIndex			: UDINT;
	ExitItemInSorter		: ST_Item;
	ExitItemFound			: ST_ItemTemporary;
	ExitInDivert			: BOOL;
	ExitDiverting			: BOOL;
	ExitSuccess				: BOOL;
	ExitDetected			: BOOL;
	ExitComplete			: BOOL;

	UpdateIndexCounter		: DINT;

	bTest : BOOL;
	sMessage	:	STRING;
	
	st_DisplayItem		:st_Item;
	LogSorterDump		:BOOL := FALSE;
	aTestBool			:	ARRAY[0..100] OF BOOL;
	
	fb_FindDestination		: FB_FindDestination;
	fb_DefaultDestination	: FB_FindDestination;
	fb_RecircDestination	: FB_FindDestination;
	// Created to allow the aDiverts to be used in the FB_FindDestination Function Block
	aTempDiverts			: ARRAY[SorterExample.DIVERTMIN..SorterExample.NUMBEROFDIVERTS] OF ST_DIVERT;
END_VAR


aTempDiverts := aDiverts;
// Initialize the Transport and Update buffers
// Set Master for FB's that control the buffer
fb_ArrivalBuffer.Master := FALSE;
fb_TransportBuffer.Master := FALSE;
fb_UpdateBuffer.Master := TRUE;

// Turn ON/OFF Logging of all activity in/out
fb_ArrivalBuffer.LogEntries := .nItemBufferLogEnable.ARRIVALS;
fb_TransportBuffer.LogEntries := .nItemBufferLogEnable.TRANSPORT;
fb_UpdateBuffer.LogEntries := .nItemBufferLogEnable.UPDATE;

// Provide names for the buffers
fb_ArrivalBuffer.Name := 'SRT ARRIVAL';
fb_TransportBuffer.Name := 'SRT TRANSPORT';
fb_UpdateBuffer.Name := 'SRT UPDATE';

// Initialize the FB_ItemExtBuffer Instances
fb_ArrivalBuffer(st_BufferData := st_ArrivalBuffer
						, st_BufferFdbkIn := st_ArrivalFdbkIn
						, st_BufferFdbkOut => st_ArrivalFdbkOut);
fb_TransportBuffer(st_BufferData := st_TransportBuffer
						, st_BufferFdbkIn := st_TransportFdbkIn
						, st_BufferFdbkOut => st_TransportFdbkOut);
fb_UpdateBuffer(st_BufferData := st_UpdateBuffer
						, st_BufferFdbkIn := st_UpdateFdbkIn
						, st_BufferFdbkOut => st_UpdateFdbkOut);

IF GVL_IO.INIT THEN
	fb_ArrivalBuffer.Clear();
	fb_TransportBuffer.Clear();
	fb_UpdateBuffer.Clear();
END_IF
						
(*
	Set the Upper/Lower bound of relevant arrays for looping purposes
	ItemsArrayMax/Min for the sorter array slot count
*)
// Size is Max - Min + 1 to capture both extremes
ItemsArraySize := ItemsArrayMax - ItemsArrayMin + 1;

(*
 	Check for a value disagreement in the Arrival Buffer In and Out pointers to
  	determine if there is an update for an item.
	When an Item arrives, the System PLC adds it to the shared buffer and increments
	the InPointer
*)
IF st_ArrivalBuffer.nInPointer <> fb_ArrivalBuffer.OutPointer THEN
	fb_ArrivalBuffer.RemoveItem(st_ItemToReturn => st_ArrivalItem);
END_IF

// Input Item read at bar code reader from System PLC to sorter
IF st_ArrivalItem.ID <> '' THEN
	IF .nSortBufferLogEnable.BUFFER_ARRIVAL THEN
		sMessage := CONCAT(' Item: ', st_ArrivalItem.ID);
		sMessage := CONCAT(sMessage,' Pulses: ');
		sMessage := CONCAT(sMessage, UDINT_TO_STRING(st_Sorter.EncoderCounts));
		// Write to the Error List
		ADSLOGSTR( msgCtrlMask := ADSLOG_MSGTYPE_HINT OR ADSLOG_MSGTYPE_LOG
			, msgFmtStr := 'Arrival Processed: %s'
			, strArg := sMessage);
	END_IF
	// Indicate that this item did not get added to the sorter and add to the exit buffer
	//  Both as a TransportUpdate and TransportComplete message type 
	IF st_NextToInduct.Item.ID <> '' THEN
		IF .nSortBufferLogEnable.BUFFER_MISSINDUCT THEN
			sMessage := CONCAT(' Item: ', st_NextToInduct.Item.ID);
			// Write to the Error List
			ADSLOGSTR( msgCtrlMask := ADSLOG_MSGTYPE_HINT OR ADSLOG_MSGTYPE_LOG
				, msgFmtStr := 'Item Removed - Not Inducted: %s'
				, strArg := sMessage);
		END_IF
		// Transport Response
		st_NextToInduct.Item.Status := E_StatusCode.Assign_NotInducted;
		st_NextToInduct.Item.DeviceID := st_Sorter.Config.EquipID;
		st_NextToInduct.Item.MessageType := E_MessageIds.TransportResponse_25;
		fb_UpdateBuffer.AddItem(st_ItemToAdd := st_NextToInduct.Item);

		// Transport Complete
		st_NextToInduct.Item.Status := E_StatusCode.Divert_NotInducted;
		st_NextToInduct.Item.MessageType := E_MessageIds.TransportComplete_26;
		fb_UpdateBuffer.AddItem(st_ItemToAdd := st_NextToInduct.Item);
	END_IF
	// Copy Last BCR item to Item to Induct
	st_NextToInduct.Item :=  st_ArrivalItem;
	// Add the Sorter EquipID to the NextToInduct
	st_NextToInduct.Item.DeviceID := st_Sorter.Config.EquipID;
	// Set the Default Destination
	st_NextToInduct.Item.Destination := st_Sorter.Config.DefaultDestination;
	// Capture an encoder value that when the encoder count exceeds this value, NextToInduct item will be cleared
	st_NextToInduct.Counts := st_Sorter.EncoderCounts;
	// Clear the Last recieved item
	st_ArrivalItem := BlankItem;
	// Prepare to replace the Temporarily assigned item with this item
	IF st_TempInductItem.Item.ID <> '' THEN
		// Capture the Counts and Length from the temporary item
		st_NextToInduct.Counts := st_TempInductItem.Counts;
		st_NextToInduct.Item.Length := st_TempInductItem.Item.Length;
		//Identify the Item to replace in the sorter array
		st_ReplaceItem := st_TempInductItem.Item;
		st_TempInductItem.Counts := 0;
		st_TempInductItem.Item := BlankItem;
		IF .nSortBufferLogEnable.BUFFER_TEMPINDUCT THEN
			ADSLOGSTR( msgCtrlMask := ADSLOG_MSGTYPE_HINT OR ADSLOG_MSGTYPE_LOG
				, msgFmtStr := 'Temp ID Replaced : %s'
				, strArg := st_ReplaceItem.ID); 
		END_IF
	END_IF
END_IF

(*
 	Check for a value disagreement in the SorterTransportBuffer In and Out pointers to
  	determine if there is an update for an item.
	When an update arrived, the System PLC adds it to the shared buffer and increments
	the InPointer
*)
IF st_TransportBuffer.nInPointer <> fb_TransportBuffer.OutPointer THEN
	fb_TransportBuffer.RemoveItem(st_ItemToReturn => st_ToUpdate.Item);
	// Lookup the index for the chosen destination
	fb_FindDestination(RoundRobin := st_Sorter.Config.RoundRobin
					, aDiverts := aTempDiverts
					, DestinationID := st_ToUpdate.Item.Destination
					, DestinationIndex => st_ToUpdate.Item.DestinationIdx);
	IF .nSortBufferLogEnable.BUFFER_DESTINDEX THEN
		sMessage := CONCAT(' Item: ', st_ToUpdate.Item.ID);
		sMessage := CONCAT(sMessage,' Destination: ');
		sMessage := CONCAT(sMessage, UDINT_TO_STRING(TransportSorterIndex));
		sMessage := CONCAT(sMessage,' Index: ');
		sMessage := CONCAT(sMessage, UDINT_TO_STRING(TransportSorterIndex));
		// Write to the Error List
		ADSLOGSTR( msgCtrlMask := ADSLOG_MSGTYPE_HINT OR ADSLOG_MSGTYPE_LOG
			, msgFmtStr := 'Divert Index of Destination: %s'
			, strArg := sMessage);
	END_IF
END_IF

// Get the Default Destination Index
fb_DefaultDestination(RoundRobin := st_Sorter.Config.RoundRobin
				, aDiverts := aTempDiverts
				, DestinationID := st_Sorter.Config.DefaultDestination
				, DestinationIndex => st_Sorter.Config.DefaultDestIdx);

// Get the Recirculation Destination Index
fb_RecircDestination(RoundRobin := st_Sorter.Config.RoundRobin
				, aDiverts := aTempDiverts
				, DestinationID := st_Sorter.Config.RecircDestination
				, DestinationIndex => st_Sorter.Config.RecircDestIdx);

// Test the Item to Update against the Item to Induct and update if they match:
//	Update the NextItemToInduct with the updated data, then clear the Item to Update
IF st_ToUpdate.Item.ID <> '' THEN
	IF st_ToUpdate.Item.ID = st_NextToInduct.Item.ID THEN
		// Indicate that the transport command was received and a response was sent
		st_NextToInduct.Item.MessageType := E_MessageIds.TransportResponse_25;
		// Test the assigned lane for availability
		IF aDiverts[st_ToUpdate.Item.DestinationIdx].Full
		   OR aDiverts[st_ToUpdate.Item.DestinationIdx].Faulted THEN
			// Prepare a message to indicate that the item cannot be assigned
			st_ToUpdate.Item.Status := E_StatusCode.Assign_Full;
			st_ToUpdate.Item.DeviceID := st_Sorter.Config.EquipID;
			st_ToUpdate.Item.MessageType := E_MessageIds.TransportResponse_25;
			fb_UpdateBuffer.AddItem(st_ItemToAdd := st_ToUpdate.Item);
			st_NextToInduct.Item.ExtStatus := E_StatusCode.Divert_Full;
		ELSE
			st_NextToInduct.Item.DeviceID := st_Sorter.Config.EquipID;
			st_NextToInduct.Item.Status := E_StatusCode.Assign_Accepted;
			// Update the Destination
			st_NextToInduct.Item.Destination := st_ToUpdate.Item.Destination;
			st_NextToInduct.Item.DestinationIdx := st_ToUpdate.Item.DestinationIdx;
			fb_UpdateBuffer.AddItem(st_ItemToAdd := st_NextToInduct.Item);
		END_IF
		// If commissioning, ignore any other direction
		IF DivertToCommission > 0 THEN
			st_NextToInduct.Item.Destination := DivertToCommission;
		END_IF
		// Log the update
		IF .nSortBufferLogEnable.BUFFER_INDUCT THEN
			sMessage := CONCAT(' Item: ', st_ToUpdate.Item.ID);
			sMessage := CONCAT(sMessage,' Pulses: ');
			sMessage := CONCAT(sMessage, UDINT_TO_STRING(st_Sorter.EncoderCounts));
			sMessage := CONCAT(sMessage,' Status: ');
			sMessage := CONCAT(sMessage, UDINT_TO_STRING(st_ToUpdate.Item.Status));
			sMessage := CONCAT(sMessage,' Ext Status: ');
			sMessage := CONCAT(sMessage, UDINT_TO_STRING(st_ToUpdate.Item.ExtStatus));
			// Write to the Error List
			ADSLOGSTR( msgCtrlMask := ADSLOG_MSGTYPE_HINT OR ADSLOG_MSGTYPE_LOG
				, msgFmtStr := 'Found Before Induct: %s'
				, strArg := sMessage);
		END_IF
		// We updated the item we were inducting, clear the Item to update
		st_ToUpdate.Item := BlankItem;
	END_IF
END_IF

// Clear the Update Item Found record each pass
TransportItemFound := BlankItem;

// Clear the last detected Exit item
ExitItemFound.Item := BlankItem;

// Reset the Detection booleans
ExitInDivert := FALSE;
ExitDiverting := FALSE;
ExitDetected := FALSE;
ExitSuccess := FALSE;
ExitComplete := FALSE;

// Loop through the entire array, it should be appropriately sized for the length of the sorter section
FOR UpdateIndexCounter := UDINT_TO_DINT(ItemsArrayMin) TO UDINT_TO_DINT(ItemsArrayMax) DO //Loop through everything in the sorter	

	// For Transport commands, start from the current encoder count and work forwards, just like the exit
	TransportSorterIndex := F_CalculateIndex(Offset := (UpdateIndexCounter)
											, InitialValue := st_Sorter.EncoderCounts
											, BufferSize := ItemsArraySize);

	// This is the item in the sorter array that we will be procesing this pass, testing for a Transport update message
	TransportItemInSorter := aItems[UDINT_TO_DINT(TransportSorterIndex)];

	// Test for a replace item
	// ReplaceItem is the temporary item
	// NextToInduct is the item to replace the temporary with
	IF st_ReplaceItem.ID <> '' THEN
		IF st_ReplaceItem.ID = TransportItemInSorter.ID THEN
			IF .nSortBufferLogEnable.BUFFER_REPLACEINDUCT THEN
				sMessage := CONCAT(' Item: ', st_ReplaceItem.ID);
				sMessage := CONCAT(sMessage,' New Item: ');
				sMessage := CONCAT(sMessage, st_NextToInduct.Item.ID);
				sMessage := CONCAT(sMessage,' Index: ');
				sMessage := CONCAT(sMessage, UDINT_TO_STRING(TransportSorterIndex));
				sMessage := CONCAT(sMessage,' Orig Dest: ');
				sMessage := CONCAT(sMessage, DINT_TO_STRING(TransportItemInSorter.Destination));
				sMessage := CONCAT(sMessage,' New Dest: ');
				sMessage := CONCAT(sMEssage, DINT_TO_STRING(st_ReplaceItem.Destination));
				// Write to the Error List
				ADSLOGSTR( msgCtrlMask := ADSLOG_MSGTYPE_HINT OR ADSLOG_MSGTYPE_LOG
					, msgFmtStr := 'Item ID Replaced After Induct: %s'
					, strArg := sMessage);
			END_IF
			TransportItemInSorter.ID := st_NextToInduct.Item.ID;
			TransportItemInSorter.Destination := st_NextToInduct.Item.Destination;
			TransportItemInSorter.DeviceID := st_NextToInduct.Item.DeviceID;
			TransportItemInSorter.MessageType := st_NextToInduct.Item.MessageType;
			TransportItemInSorter.Status := st_NextToInduct.Item.Status;
			TransportItemInSorter.UniqueID := st_NextToInduct.Item.UniqueID;
			TransportItemInSorter.CapturedInMetrics := st_NextToInduct.Item.CapturedInMetrics;
		END_IF
	END_IF
	// Test for an Item Update
	IF st_ToUpdate.Item.ID <> '' THEN
		// Test the sorter item against the update item
		IF st_ToUpdate.Item.ID = TransportItemInSorter.ID THEN
			IF .nSortBufferLogEnable.BUFFER_UPDATEINDUCT THEN
				sMessage := CONCAT(' Item: ', st_ToUpdate.Item.ID);
				sMessage := CONCAT(sMessage,' Index: ');
				sMessage := CONCAT(sMessage, UDINT_TO_STRING(TransportSorterIndex));
				// Write to the Error List
				ADSLOGSTR( msgCtrlMask := ADSLOG_MSGTYPE_HINT OR ADSLOG_MSGTYPE_LOG
					, msgFmtStr := 'Found After Induct: %s'
					, strArg := sMessage);
			END_IF
			// Copy the found item record, 
			TransportItemFound := TransportItemInSorter;
			// Test the destined divert for availability
			IF aDiverts[st_ToUpdate.Item.DestinationIdx].Full OR aDiverts[st_ToUpdate.Item.DestinationIdx].Faulted THEN
				// Prepare a message to indicate that the item cannot be assigned
				TransportItemFound.Status := E_StatusCode.Assign_Full;
				TransportItemFound.ExtStatus := E_StatusCode.Divert_Full;
				TransportItemFound.MessageType := E_MessageIds.TransportResponse_25;
				TransportItemFound.Destination := st_Sorter.Config.DefaultDestination;
				TransportItemFound.DestinationIdx := st_Sorter.Config.DefaultDestIdx;
			// Test for an already diverting item and assign an ExtStatus of LateAssignment
			ELSIF TransportItemInSorter.Status >= E_StatusCode.Diverting THEN
				TransportItemFound.ExtStatus := E_StatusCode.Divert_LateAssignment;
				TransportItemFound.MessageType := E_MessageIds.TransportResponse_25;
			ELSE
				//  Change the destination, which should be the only item in the update
				TransportItemFound.Destination := st_ToUpdate.Item.Destination;
				TransportItemFound.DestinationIdx := st_ToUpdate.Item.DestinationIdx;
				// This message indicates we could assign the Item
				TransportItemFound.Status := E_StatusCode.Assign_Accepted;
				TransportItemFound.MessageType := E_MessageIds.TransportResponse_25;
			END_IF
			TransportItemFound.DeviceID := st_Sorter.Config.EquipID;
			// Add the item to the update buffer
			fb_UpdateBuffer.AddItem(TransportItemFound);
			// Clear the ToUpdate Item
			st_ToUpdate.Item := BlankItem;
		END_IF
	END_IF
	
